	W =180.000 deg,	P =   0.000 deg,	R =    90.000 deg
};
P[5219]{
   GP1:
	UF : 1, UT : 1,		CONFIG : 'N U T, 0, 0, 1',
	X =  91.000  mm,	Y =  97.000  mm,	Z =   0.600 mm,
	W =180.000 deg,	P =   0.000 deg,	R =    90.000 deg
};
P[5220]{
   GP1:
	UF : 1, UT : 1,		CONFIG : 'N U T, 0, 0, 1',
	X =  91.000  mm,	Y =  97.000  mm,	Z =   15.000 mm,
	W =180.000 deg,	P =   0.000 deg,	R =    90.000 deg
};
P[5221]{
   GP1:
	UF : 1, UT : 1,		CONFIG : 'N U T, 0, 0, 1',
	X =  94.000  mm,	Y =  97.000  mm,	Z =   15.000 mm,
	W =180.000 deg,	P =   0.000 deg,	R =    90.000 deg
};
P[5222]{
   GP1:
	UF : 1, UT : 1,		CONFIG : 'N U T, 0, 0, 1',
	X =  94.000  mm,	Y =  97.000  mm,	Z =   0.600 mm,
	W =180.000 deg,	P =   0.000 deg,	R =    90.000 deg
};
P[5223]{
   GP1:
	UF : 1, UT : 1,		CONFIG : 'N U T, 0, 0, 1',
	X =  94.000  mm,	Y =  97.000  mm,	Z =   15.000 mm,
	W =180.000 deg,	P =   0.000 deg,	R =    90.000 deg
};
P[5224]{
   GP1:
	UF : 1, UT : 1,		CONFIG : 'N U T, 0, 0, 1',
	X =  97.000  mm,	Y =  97.000  mm,	Z =   15.000 mm,
	W =180.000 deg,	P =   0.000 deg,	R =    90.000 deg
};
P[5225]{
   GP1:
	UF : 1, UT : 1,		CONFIG : 'N U T, 0, 0, 1',
	X =  97.000  mm,	Y =  97.000  mm,	Z =   0.600 mm,
	W =180.000 deg,	P =   0.000 deg,	R =    90.000 deg
};
P[5226]{
   GP1:
	UF : 1, UT : 1,		CONFIG : 'N U T, 0, 0, 1',
	X =  97.000  mm,	Y =  97.000  mm,	Z =   15.000 mm,
	W =180.000 deg,	P =   0.000 deg,	R =    90.000 deg
};
P[5227]{
   GP1:
	UF : 1, UT : 1,		CONFIG : 'N U T, 0, 0, 1',
	X =  100.000  mm,	Y =  97.000  mm,	Z =   15.000 mm,
	W =180.000 deg,	P =   0.000 deg,	R =    90.000 deg
};
P[5228]{
   GP1:
	UF : 1, UT : 1,		CONFIG : 'N U T, 0, 0, 1',
	X =  100.000  mm,	Y =  97.000  mm,	Z =   0.600 mm,
	W =180.000 deg,	P =   0.000 deg,	R =    90.000 deg
};
P[5229]{
   GP1:
	UF : 1, UT : 1,		CONFIG : 'N U T, 0, 0, 1',
	X =  100.000  mm,	Y =  97.000  mm,	Z =   15.000 mm,
	W =180.000 deg,	P =   0.000 deg,	R =    90.000 deg
};
P[5230]{
   GP1:
	UF : 1, UT : 1,		CONFIG : 'N U T, 0, 0, 1',
	X =  103.000  mm,	Y =  97.000  mm,	Z =   15.000 mm,
	W =180.000 deg,	P =   0.000 deg,	R =    90.000 deg
};
P[5231]{
   GP1:
	UF : 1, UT : 1,		CONFIG : 'N U T, 0, 0, 1',
	X =  103.000  mm,	Y =  97.000  mm,	Z =   0.600 mm,
	W =180.000 deg,	P =   0.000 deg,	R =    90.000 deg
};
P[5232]{
   GP1:
	UF : 1, UT : 1,		CONFIG : 'N U T, 0, 0, 1',
	X =  103.000  mm,	Y =  97.000  mm,	Z =   15.000 mm,
	W =180.000 deg,	P =   0.000 deg,	R =    90.000 deg
};
P[5233]{
   GP1:
	UF : 1, UT : 1,		CONFIG : 'N U T, 0, 0, 1',
	X =  106.000  mm,	Y =  97.000  mm,	Z =   15.000 mm,
	W =180.000 deg,	P =   0.000 deg,	R =    90.000 deg
};
P[5234]{
   GP1:
	UF : 1, UT : 1,		CONFIG : 'N U T, 0, 0, 1',
	X =  106.000  mm,	Y =  97.000  mm,	Z =   0.600 mm,
	W =180.000 deg,	P =   0.000 deg,	R =    90.000 deg
};
P[5235]{
   GP1:
	UF : 1, UT : 1,		CONFIG : 'N U T, 0, 0, 1',
	X =  106.000  mm,	Y =  97.000  mm,	Z =   15.000 mm,
	W =180.000 deg,	P =   0.000 deg,	R =    90.000 deg
};
P[5236]{
   GP1:
	UF : 1, UT : 1,		CONFIG : 'N U T, 0, 0, 1',
	X =  109.000  mm,	Y =  97.000  mm,	Z =   15.000 mm,
	W =180.000 deg,	P =   0.000 deg,	R =    90.000 deg
};
P[5237]{
   GP1:
	UF : 1, UT : 1,		CONFIG : 'N U T, 0, 0, 1',
	X =  109.000  mm,	Y =  97.000  mm,	Z =   0.600 mm,
	W =180.000 deg,	P =   0.000 deg,	R =    90.000 deg
};
P[5238]{
   GP1:
	UF : 1, UT : 1,		CONFIG : 'N U T, 0, 0, 1',
	X =  109.000  mm,	Y =  97.000  mm,	Z =   15.000 mm,
	W =180.000 deg,	P =   0.000 deg,	R =    90.000 deg
};
P[5239]{
   GP1:
	UF : 1, UT : 1,		CONFIG : 'N U T, 0, 0, 1',
	X =  112.000  mm,	Y =  97.000  mm,	Z =   15.000 mm,
	W =180.000 deg,	P =   0.000 deg,	R =    90.000 deg
};
P[5240]{
   GP1:
	UF : 1, UT : 1,		CONFIG : 'N U T, 0, 0, 1',
	X =  112.000  mm,	Y =  97.000  mm,	Z =   0.600 mm,
	W =180.000 deg,	P =   0.000 deg,	R =    90.000 deg
};
P[5241]{
   GP1:
	UF : 1, UT : 1,		CONFIG : 'N U T, 0, 0, 1',
	X =  112.000  mm,	Y =  97.000  mm,	Z =   15.000 mm,
	W =180.000 deg,	P =   0.000 deg,	R =    90.000 deg
};
P[5242]{
   GP1:
	UF : 1, UT : 1,		CONFIG : 'N U T, 0, 0, 1',
	X =  115.000  mm,	Y =  97.000  mm,	Z =   15.000 mm,
	W =180.000 deg,	P =   0.000 deg,	R =    90.000 deg
};
P[5243]{
   GP1:
	UF : 1, UT : 1,		CONFIG : 'N U T, 0, 0, 1',
	X =  115.000  mm,	Y =  97.000  mm,	Z =   0.600 mm,
	W =180.000 deg,	P =   0.000 deg,	R =    90.000 deg
};
P[5244]{
   GP1:
	UF : 1, UT : 1,		CONFIG : 'N U T, 0, 0, 1',
	X =  115.000  mm,	Y =  97.000  mm,	Z =   15.000 mm,
	W =180.000 deg,	P =   0.000 deg,	R =    90.000 deg
};
P[5260]{
   GP1:
	UF : 1, UT : 1,		CONFIG : 'N U T, 0, 0, 1',
	X =  133.000  mm,	Y =  97.000  mm,	Z =   15.000 mm,
	W =180.000 deg,	P =   0.000 deg,	R =    90.000 deg
};
P[5261]{
   GP1:
	UF : 1, UT : 1,		CONFIG : 'N U T, 0, 0, 1',
	X =  133.000  mm,	Y =  97.000  mm,	Z =   0.600 mm,
	W =180.000 deg,	P =   0.000 deg,	R =    90.000 deg
};
P[5262]{
   GP1:
	UF : 1, UT : 1,		CONFIG : 'N U T, 0, 0, 1',
	X =  133.000  mm,	Y =  97.000  mm,	Z =   15.000 mm,
	W =180.000 deg,	P =   0.000 deg,	R =    90.000 deg
};
P[5263]{
   GP1:
	UF : 1, UT : 1,		CONFIG : 'N U T, 0, 0, 1',
	X =  136.000  mm,	Y =  97.000  mm,	Z =   15.000 mm,
	W =180.000 deg,	P =   0.000 deg,	R =    90.000 deg
};
P[5264]{
   GP1:
	UF : 1, UT : 1,		CONFIG : 'N U T, 0, 0, 1',
	X =  136.000  mm,	Y =  97.000  mm,	Z =   0.600 mm,
	W =180.000 deg,	P =   0.000 deg,	R =    90.000 deg
};
P[5265]{
   GP1:
	UF : 1, UT : 1,		CONFIG : 'N U T, 0, 0, 1',
	X =  136.000  mm,	Y =  97.000  mm,	Z =   15.000 mm,
	W =180.000 deg,	P =   0.000 deg,	R =    90.000 deg
};
P[5266]{
   GP1:
	UF : 1, UT : 1,		CONFIG : 'N U T, 0, 0, 1',
	X =  139.000  mm,	Y =  97.000  mm,	Z =   15.000 mm,
	W =180.000 deg,	P =   0.000 deg,	R =    90.000 deg
};
P[5267]{
   GP1:
	UF : 1, UT : 1,		CONFIG : 'N U T, 0, 0, 1',
	X =  139.000  mm,	Y =  97.000  mm,	Z =   0.600 mm,
	W =180.000 deg,	P =   0.000 deg,	R =    90.000 deg
};
P[5268]{
   GP1:
	UF : 1, UT : 1,		CONFIG : 'N U T, 0, 0, 1',
	X =  139.000  mm,	Y =  97.000  mm,	Z =   15.000 mm,
	W =180.000 deg,	P =   0.000 deg,	R =    90.000 deg
};
P[5278]{
   GP1:
	UF : 1, UT : 1,		CONFIG : 'N U T, 0, 0, 1',
	X =  163.000  mm,	Y =  97.000  mm,	Z =   15.000 mm,
	W =180.000 deg,	P =   0.000 deg,	R =    90.000 deg
};
P[5279]{
   GP1:
	UF : 1, UT : 1,		CONFIG : 'N U T, 0, 0, 1',
	X =  163.000  mm,	Y =  97.000  mm,	Z =   0.600 mm,
	W =180.000 deg,	P =   0.000 deg,	R =    90.000 deg
};
P[5280]{
   GP1:
	UF : 1, UT : 1,		CONFIG : 'N U T, 0, 0, 1',
	X =  163.000  mm,	Y =  97.000  mm,	Z =   15.000 mm,
	W =180.000 deg,	P =   0.000 deg,	R =    90.000 deg
};
P[5281]{
   GP1:
	UF : 1, UT : 1,		CONFIG : 'N U T, 0, 0, 1',
	X =  166.000  mm,	Y =  97.000  mm,	Z =   15.000 mm,
	W =180.000 deg,	P =   0.000 deg,	R =    90.000 deg
};
P[5282]{
   GP1:
	UF : 1, UT : 1,		CONFIG : 'N U T, 0, 0, 1',
	X =  166.000  mm,	Y =  97.000  mm,	Z =   0.600 mm,
	W =180.000 deg,	P =   0.000 deg,	R =    90.000 deg
};
P[5283]{
   GP1:
	UF : 1, UT : 1,		CONFIG : 'N U T, 0, 0, 1',
	X =  166.000  mm,	Y =  97.000  mm,	Z =   15.000 mm,
	W =180.000 deg,	P =   0.000 deg,	R =    90.000 deg
};
P[5284]{
   GP1:
	UF : 1, UT : 1,		CONFIG : 'N U T, 0, 0, 1',
	X =  169.000  mm,	Y =  97.000  mm,	Z =   15.000 mm,
	W =180.000 deg,	P =   0.000 deg,	R =    90.000 deg
};
P[5285]{
   GP1:
	UF : 1, UT : 1,		CONFIG : 'N U T, 0, 0, 1',
	X =  169.000  mm,	Y =  97.000  mm,	Z =   0.600 mm,
	W =180.000 deg,	P =   0.000 deg,	R =    90.000 deg
};
P[5286]{
   GP1:
	UF : 1, UT : 1,		CONFIG : 'N U T, 0, 0, 1',
	X =  169.000  mm,	Y =  97.000  mm,	Z =   15.000 mm,
	W =180.000 deg,	P =   0.000 deg,	R =    90.000 deg
};
P[5287]{
   GP1:
	UF : 1, UT : 1,		CONFIG : 'N U T, 0, 0, 1',
	X =  172.000  mm,	Y =  97.000  mm,	Z =   15.000 mm,
	W =180.000 deg,	P =   0.000 deg,	R =    90.000 deg
};
P[5288]{
   GP1:
	UF : 1, UT : 1,		CONFIG : 'N U T, 0, 0, 1',
	X =  172.000  mm,	Y =  97.000  mm,	Z =   0.600 mm,
	W =180.000 deg,	P =   0.000 deg,	R =    90.000 deg
};
P[5289]{
   GP1:
	UF : 1, UT : 1,		CONFIG : 'N U T, 0, 0, 1',
	X =  172.000  mm,	Y =  97.000  mm,	Z =   15.000 mm,
	W =180.000 deg,	P =   0.000 deg,	R =    90.000 deg
};
P[5290]{
   GP1:
	UF : 1, UT : 1,		CONFIG : 'N U T, 0, 0, 1',
	X =  175.000  mm,	Y =  97.000  mm,	Z =   15.000 mm,
	W =180.000 deg,	P =   0.000 deg,	R =    90.000 deg
};
P[5291]{
   GP1:
	UF : 1, UT : 1,		CONFIG : 'N U T, 0, 0, 1',
	X =  175.000  mm,	Y =  97.000  mm,	Z =   0.600 mm,
	W =180.000 deg,	P =   0.000 deg,	R =    90.000 deg
};
P[5292]{
   GP1:
	UF : 1, UT : 1,		CONFIG : 'N U T, 0, 0, 1',
	X =  175.000  mm,	Y =  97.000  mm,	Z =   15.000 mm,
	W =180.000 deg,	P =   0.000 deg,	R =    90.000 deg
};
P[5293]{
   GP1:
	UF : 1, UT : 1,		CONFIG : 'N U T, 0, 0, 1',
	X =  178.000  mm,	Y =  97.000  mm,	Z =   15.000 mm,
	W =180.000 deg,	P =   0.000 deg,	R =    90.000 deg
};
P[5294]{
   GP1:
	UF : 1, UT : 1,		CONFIG : 'N U T, 0, 0, 1',
	X =  178.000  mm,	Y =  97.000  mm,	Z =   0.600 mm,
	W =180.000 deg,	P =   0.000 deg,	R =    90.000 deg
};
P[5295]{
   GP1:
	UF : 1, UT : 1,		CONFIG : 'N U T, 0, 0, 1',
	X =  178.000  mm,	Y =  97.000  mm,	Z =   15.000 mm,
	W =180.000 deg,	P =   0.000 deg,	R =    90.000 deg
};
P[5299]{
   GP1:
	UF : 1, UT : 1,		CONFIG : 'N U T, 0, 0, 1',
	X =  4.000  mm,	Y =  100.000  mm,	Z =   15.000 mm,
	W =180.000 deg,	P =   0.000 deg,	R =    90.000 deg
};
P[5300]{
   GP1:
	UF : 1, UT : 1,		CONFIG : 'N U T, 0, 0, 1',
	X =  4.000  mm,	Y =  100.000  mm,	Z =   0.600 mm,
	W =180.000 deg,	P =   0.000 deg,	R =    90.000 deg
};
P[5301]{
   GP1:
	UF : 1, UT : 1,		CONFIG : 'N U T, 0, 0, 1',
	X =  4.000  mm,	Y =  100.000  mm,	Z =   15.000 mm,
	W =180.000 deg,	P =   0.000 deg,	R =    90.000 deg
};
P[5305]{
   GP1:
	UF : 1, UT : 1,		CONFIG : 'N U T, 0, 0, 1',
	X =  10.000  mm,	Y =  100.000  mm,	Z =   15.000 mm,
	W =180.000 deg,	P =   0.000 deg,	R =    90.000 deg
};
P[5306]{
   GP1:
	UF : 1, UT : 1,		CONFIG : 'N U T, 0, 0, 1',
	X =  10.000  mm,	Y =  100.000  mm,	Z =   0.600 mm,
	W =180.000 deg,	P =   0.000 deg,	R =    90.000 deg
};
P[5307]{
   GP1:
	UF : 1, UT : 1,		CONFIG : 'N U T, 0, 0, 1',
	X =  10.000  mm,	Y =  100.000  mm,	Z =   15.000 mm,
	W =180.000 deg,	P =   0.000 deg,	R =    90.000 deg
};
P[5308]{
   GP1:
	UF : 1, UT : 1,		CONFIG : 'N U T, 0, 0, 1',
	X =  13.000  mm,	Y =  100.000  mm,	Z =   15.000 mm,
	W =180.000 deg,	P =   0.000 deg,	R =    90.000 deg
};
P[5309]{
   GP1:
	UF : 1, UT : 1,		CONFIG : 'N U T, 0, 0, 1',
	X =  13.000  mm,	Y =  100.000  mm,	Z =   0.600 mm,
	W =180.000 deg,	P =   0.000 deg,	R =    90.000 deg
};
P[5310]{
   GP1:
	UF : 1, UT : 1,		CONFIG : 'N U T, 0, 0, 1',
	X =  13.000  mm,	Y =  100.000  mm,	Z =   15.000 mm,
	W =180.000 deg,	P =   0.000 deg,	R =    90.000 deg
};
P[5320]{
   GP1:
	UF : 1, UT : 1,		CONFIG : 'N U T, 0, 0, 1',
	X =  25.000  mm,	Y =  100.000  mm,	Z =   15.000 mm,
	W =180.000 deg,	P =   0.000 deg,	R =    90.000 deg
};
P[5321]{
   GP1:
	UF : 1, UT : 1,		CONFIG : 'N U T, 0, 0, 1',
	X =  25.000  mm,	Y =  100.000  mm,	Z =   0.600 mm,
	W =180.000 deg,	P =   0.000 deg,	R =    90.000 deg
};
P[5322]{
   GP1:
	UF : 1, UT : 1,		CONFIG : 'N U T, 0, 0, 1',
	X =  25.000  mm,	Y =  100.000  mm,	Z =   15.000 mm,
	W =180.000 deg,	P =   0.000 deg,	R =    90.000 deg
};
P[5323]{
   GP1:
	UF : 1, UT : 1,		CONFIG : 'N U T, 0, 0, 1',
	X =  28.000  mm,	Y =  100.000  mm,	Z =   15.000 mm,
	W =180.000 deg,	P =   0.000 deg,	R =    90.000 deg
};
P[5324]{
   GP1:
	UF : 1, UT : 1,		CONFIG : 'N U T, 0, 0, 1',
	X =  28.000  mm,	Y =  100.000  mm,	Z =   0.600 mm,
	W =180.000 deg,	P =   0.000 deg,	R =    90.000 deg
};
P[5325]{
   GP1:
	UF : 1, UT : 1,		CONFIG : 'N U T, 0, 0, 1',
	X =  28.000  mm,	Y =  100.000  mm,	Z =   15.000 mm,
	W =180.000 deg,	P =   0.000 deg,	R =    90.000 deg
};
P[5335]{
   GP1:
	UF : 1, UT : 1,		CONFIG : 'N U T, 0, 0, 1',
	X =  40.000  mm,	Y =  100.000  mm,	Z =   15.000 mm,
	W =180.000 deg,	P =   0.000 deg,	R =    90.000 deg
};
P[5336]{
   GP1:
	UF : 1, UT : 1,		CONFIG : 'N U T, 0, 0, 1',
	X =  40.000  mm,	Y =  100.000  mm,	Z =   0.600 mm,
	W =180.000 deg,	P =   0.000 deg,	R =    90.000 deg
};
P[5337]{
   GP1:
	UF : 1, UT : 1,		CONFIG : 'N U T, 0, 0, 1',
	X =  40.000  mm,	Y =  100.000  mm,	Z =   15.000 mm,
	W =180.000 deg,	P =   0.000 deg,	R =    90.000 deg
};
P[5338]{
   GP1:
	UF : 1, UT : 1,		CONFIG : 'N U T, 0, 0, 1',
	X =  43.000  mm,	Y =  100.000  mm,	Z =   15.000 mm,
	W =180.000 deg,	P =   0.000 deg,	R =    90.000 deg
};
P[5339]{
   GP1:
	UF : 1, UT : 1,		CONFIG : 'N U T, 0, 0, 1',
	X =  43.000  mm,	Y =  100.000  mm,	Z =   0.600 mm,
	W =180.000 deg,	P =   0.000 deg,	R =    90.000 deg
};
P[5340]{
   GP1:
	UF : 1, UT : 1,		CONFIG : 'N U T, 0, 0, 1',
	X =  43.000  mm,	Y =  100.000  mm,	Z =   15.000 mm,
	W =180.000 deg,	P =   0.000 deg,	R =    90.000 deg
};
P[5341]{
   GP1:
	UF : 1, UT : 1,		CONFIG : 'N U T, 0, 0, 1',
	X =  46.000  mm,	Y =  100.000  mm,	Z =   15.000 mm,
	W =180.000 deg,	P =   0.000 deg,	R =    90.000 deg
};
P[5342]{
   GP1:
	UF : 1, UT : 1,		CONFIG : 'N U T, 0, 0, 1',
	X =  46.000  mm,	Y =  100.000  mm,	Z =   0.600 mm,
	W =180.000 deg,	P =   0.000 deg,	R =    90.000 deg
};
P[5343]{
   GP1:
	UF : 1, UT : 1,		CONFIG : 'N U T, 0, 0, 1',
	X =  46.000  mm,	Y =  100.000  mm,	Z =   15.000 mm,
	W =180.000 deg,	P =   0.000 deg,	R =    90.000 deg
};
P[5344]{
   GP1:
	UF : 1, UT : 1,		CONFIG : 'N U T, 0, 0, 1',
	X =  49.000  mm,	Y =  100.000  mm,	Z =   15.000 mm,
	W =180.000 deg,	P =   0.000 deg,	R =    90.000 deg
};
P[5345]{
   GP1:
	UF : 1, UT : 1,		CONFIG : 'N U T, 0, 0, 1',
	X =  49.000  mm,	Y =  100.000  mm,	Z =   0.600 mm,
	W =180.000 deg,	P =   0.000 deg,	R =    90.000 deg
};
P[5346]{
   GP1:
	UF : 1, UT : 1,		CONFIG : 'N U T, 0, 0, 1',
	X =  49.000  mm,	Y =  100.000  mm,	Z =   15.000 mm,
	W =180.000 deg,	P =   0.000 deg,	R =    90.000 deg
};
P[5347]{
   GP1:
	UF : 1, UT : 1,		CONFIG : 'N U T, 0, 0, 1',
	X =  52.000  mm,	Y =  100.000  mm,	Z =   15.000 mm,
	W =180.000 deg,	P =   0.000 deg,	R =    90.000 deg
};
P[5348]{
   GP1:
	UF : 1, UT : 1,		CONFIG : 'N U T, 0, 0, 1',
	X =  52.000  mm,	Y =  100.000  mm,	Z =   0.600 mm,
	W =180.000 deg,	P =   0.000 deg,	R =    90.000 deg
};
P[5349]{
   GP1:
	UF : 1, UT : 1,		CONFIG : 'N U T, 0, 0, 1',
	X =  52.000  mm,	Y =  100.000  mm,	Z =   15.000 mm,
	W =180.000 deg,	P =   0.000 deg,	R =    90.000 deg
};
P[5350]{
   GP1:
	UF : 1, UT : 1,		CONFIG : 'N U T, 0, 0, 1',
	X =  55.000  mm,	Y =  100.000  mm,	Z =   15.000 mm,
	W =180.000 deg,	P =   0.000 deg,	R =    90.000 deg
};
P[5351]{
   GP1:
	UF : 1, UT : 1,		CONFIG : 'N U T, 0, 0, 1',
	X =  55.000  mm,	Y =  100.000  mm,	Z =   0.600 mm,
	W =180.000 deg,	P =   0.000 deg,	R =    90.000 deg
};
P[5352]{
   GP1:
	UF : 1, UT : 1,		CONFIG : 'N U T, 0, 0, 1',
	X =  55.000  mm,	Y =  100.000  mm,	Z =   15.000 mm,
	W =180.000 deg,	P =   0.000 deg,	R =    90.000 deg
};
P[5356]{
   GP1:
	UF : 1, UT : 1,		CONFIG : 'N U T, 0, 0, 1',
	X =  61.000  mm,	Y =  100.000  mm,	Z =   15.000 mm,
	W =180.000 deg,	P =   0.000 deg,	R =    90.000 deg
};
P[5357]{
   GP1:
	UF : 1, UT : 1,		CONFIG : 'N U T, 0, 0, 1',
	X =  61.000  mm,	Y =  100.000  mm,	Z =   0.600 mm,
	W =180.000 deg,	P =   0.000 deg,	R =    90.000 deg
};
P[5358]{
   GP1:
	UF : 1, UT : 1,		CONFIG : 'N U T, 0, 0, 1',
	X =  61.000  mm,	Y =  100.000  mm,	Z =   15.000 mm,
	W =180.000 deg,	P =   0.000 deg,	R =    90.000 deg
};
P[5386]{
   GP1:
	UF : 1, UT : 1,		CONFIG : 'N U T, 0, 0, 1',
	X =  91.000  mm,	Y =  100.000  mm,	Z =   15.000 mm,
	W =180.000 deg,	P =   0.000 deg,	R =    90.000 deg
};
P[5387]{
   GP1:
	UF : 1, UT : 1,		CONFIG : 'N U T, 0, 0, 1',
	X =  91.000  mm,	Y =  100.000  mm,	Z =   0.600 mm,
	W =180.000 deg,	P =   0.000 deg,	R =    90.000 deg
};
P[5388]{
   GP1:
	UF : 1, UT : 1,		CONFIG : 'N U T, 0, 0, 1',
	X =  91.000  mm,	Y =  100.000  mm,	Z =   15.000 mm,
	W =180.000 deg,	P =   0.000 deg,	R =    90.000 deg
};
P[5389]{
   GP1:
	UF : 1, UT : 1,		CONFIG : 'N U T, 0, 0, 1',
	X =  94.000  mm,	Y =  100.000  mm,	Z =   15.000 mm,
	W =180.000 deg,	P =   0.000 deg,	R =    90.000 deg
};
P[5390]{
   GP1:
	UF : 1, UT : 1,		CONFIG : 'N U T, 0, 0, 1',
	X =  94.000  mm,	Y =  100.000  mm,	Z =   0.600 mm,
	W =180.000 deg,	P =   0.000 deg,	R =    90.000 deg
};
P[5391]{
   GP1:
	UF : 1, UT : 1,		CONFIG : 'N U T, 0, 0, 1',
	X =  94.000  mm,	Y =  100.000  mm,	Z =   15.000 mm,
	W =180.000 deg,	P =   0.000 deg,	R =    90.000 deg
};
P[5392]{
   GP1:
	UF : 1, UT : 1,		CONFIG : 'N U T, 0, 0, 1',
	X =  97.000  mm,	Y =  100.000  mm,	Z =   15.000 mm,
	W =180.000 deg,	P =   0.000 deg,	R =    90.000 deg
};
P[5393]{
   GP1:
	UF : 1, UT : 1,		CONFIG : 'N U T, 0, 0, 1',
	X =  97.000  mm,	Y =  100.000  mm,	Z =   0.600 mm,
	W =180.000 deg,	P =   0.000 deg,	R =    90.000 deg
};
P[5394]{
   GP1:
	UF : 1, UT : 1,		CONFIG : 'N U T, 0, 0, 1',
	X =  97.000  mm,	Y =  100.000  mm,	Z =   15.000 mm,
	W =180.000 deg,	P =   0.000 deg,	R =    90.000 deg
};
P[5395]{
   GP1:
	UF : 1, UT : 1,		CONFIG : 'N U T, 0, 0, 1',
	X =  100.000  mm,	Y =  100.000  mm,	Z =   15.000 mm,
	W =180.000 deg,	P =   0.000 deg,	R =    90.000 deg
};
P[5396]{
   GP1:
	UF : 1, UT : 1,		CONFIG : 'N U T, 0, 0, 1',
	X =  100.000  mm,	Y =  100.000  mm,	Z =   0.600 mm,
	W =180.000 deg,	P =   0.000 deg,	R =    90.000 deg
};
P[5397]{
   GP1:
	UF : 1, UT : 1,		CONFIG : 'N U T, 0, 0, 1',
	X =  100.000  mm,	Y =  100.000  mm,	Z =   15.000 mm,
	W =180.000 deg,	P =   0.000 deg,	R =    90.000 deg
};
P[5398]{
   GP1:
	UF : 1, UT : 1,		CONFIG : 'N U T, 0, 0, 1',
	X =  103.000  mm,	Y =  100.000  mm,	Z =   15.000 mm,
	W =180.000 deg,	P =   0.000 deg,	R =    90.000 deg
};
P[5399]{
   GP1:
	UF : 1, UT : 1,		CONFIG : 'N U T, 0, 0, 1',
	X =  103.000  mm,	Y =  100.000  mm,	Z =   0.600 mm,
	W =180.000 deg,	P =   0.000 deg,	R =    90.000 deg
};
P[5400]{
   GP1:
	UF : 1, UT : 1,		CONFIG : 'N U T, 0, 0, 1',
	X =  103.000  mm,	Y =  100.000  mm,	Z =   15.000 mm,
	W =180.000 deg,	P =   0.000 deg,	R =    90.000 deg
};
P[5401]{
   GP1:
	UF : 1, UT : 1,		CONFIG : 'N U T, 0, 0, 1',
	X =  106.000  mm,	Y =  100.000  mm,	Z =   15.000 mm,
	W =180.000 deg,	P =   0.000 deg,	R =    90.000 deg
};
P[5402]{
   GP1:
	UF : 1, UT : 1,		CONFIG : 'N U T, 0, 0, 1',
	X =  106.000  mm,	Y =  100.000  mm,	Z =   0.600 mm,
	W =180.000 deg,	P =   0.000 deg,	R =    90.000 deg
};
P[5403]{
   GP1:
	UF : 1, UT : 1,		CONFIG : 'N U T, 0, 0, 1',
	X =  106.000  mm,	Y =  100.000  mm,	Z =   15.000 mm,
	W =180.000 deg,	P =   0.000 deg,	R =    90.000 deg
};
P[5404]{
   GP1:
	UF : 1, UT : 1,		CONFIG : 'N U T, 0, 0, 1',
	X =  109.000  mm,	Y =  100.000  mm,	Z =   15.000 mm,
	W =180.000 deg,	P =   0.000 deg,	R =    90.000 deg
};
P[5405]{
   GP1:
	UF : 1, UT : 1,		CONFIG : 'N U T, 0, 0, 1',
	X =  109.000  mm,	Y =  100.000  mm,	Z =   0.600 mm,
	W =180.000 deg,	P =   0.000 deg,	R =    90.000 deg
};
P[5406]{
   GP1:
	UF : 1, UT : 1,		CONFIG : 'N U T, 0, 0, 1',
	X =  109.000  mm,	Y =  100.000  mm,	Z =   15.000 mm,
	W =180.000 deg,	P =   0.000 deg,	R =    90.000 deg
};
P[5407]{
   GP1:
	UF : 1, UT : 1,		CONFIG : 'N U T, 0, 0, 1',
	X =  112.000  mm,	Y =  100.000  mm,	Z =   15.000 mm,
	W =180.000 deg,	P =   0.000 deg,	R =    90.000 deg
};
P[5408]{
   GP1:
	UF : 1, UT : 1,		CONFIG : 'N U T, 0, 0, 1',
	X =  112.000  mm,	Y =  100.000  mm,	Z =   0.600 mm,
	W =180.000 deg,	P =   0.000 deg,	R =    90.000 deg
};
P[5409]{
   GP1:
	UF : 1, UT : 1,		CONFIG : 'N U T, 0, 0, 1',
	X =  112.000  mm,	Y =  100.000  mm,	Z =   15.000 mm,
	W =180.000 deg,	P =   0.000 deg,	R =    90.000 deg
};
P[5410]{
   GP1:
	UF : 1, UT : 1,		CONFIG : 'N U T, 0, 0, 1',
	X =  115.000  mm,	Y =  100.000  mm,	Z =   15.000 mm,
	W =180.000 deg,	P =   0.000 deg,	R =    90.000 deg
};
P[5411]{
   GP1:
	UF : 1, UT : 1,		CONFIG : 'N U T, 0, 0, 1',
	X =  115.000  mm,	Y =  100.000  mm,	Z =   0.600 mm,
	W =180.000 deg,	P =   0.000 deg,	R =    90.000 deg
};
P[5412]{
   GP1:
	UF : 1, UT : 1,		CONFIG : 'N U T, 0, 0, 1',
	X =  115.000  mm,	Y =  100.000  mm,	Z =   15.000 mm,
	W =180.000 deg,	P =   0.000 deg,	R =    90.000 deg
};
P[5413]{
   GP1:
	UF : 1, UT : 1,		CONFIG : 'N U T, 0, 0, 1',
	X =  118.000  mm,	Y =  100.000  mm,	Z =   15.000 mm,
	W =180.000 deg,	P =   0.000 deg,	R =    90.000 deg
};
P[5414]{
   GP1:
	UF : 1, UT : 1,		CONFIG : 'N U T, 0, 0, 1',
	X =  118.000  mm,	Y =  100.000  mm,	Z =   0.600 mm,
	W =180.000 deg,	P =   0.000 deg,	R =    90.000 deg
};
P[5415]{
   GP1:
	UF : 1, UT : 1,		CONFIG : 'N U T, 0, 0, 1',
	X =  118.000  mm,	Y =  100.000  mm,	Z =   15.000 mm,
	W =180.000 deg,	P =   0.000 deg,	R =    90.000 deg
};
P[5428]{
   GP1:
	UF : 1, UT : 1,		CONFIG : 'N U T, 0, 0, 1',
	X =  133.000  mm,	Y =  100.000  mm,	Z =   15.000 mm,
	W =180.000 deg,	P =   0.000 deg,	R =    90.000 deg
};
P[5429]{
   GP1:
	UF : 1, UT : 1,		CONFIG : 'N U T, 0, 0, 1',
	X =  133.000  mm,	Y =  100.000  mm,	Z =   0.600 mm,
	W =180.000 deg,	P =   0.000 deg,	R =    90.000 deg
};
P[5430]{
   GP1:
	UF : 1, UT : 1,		CONFIG : 'N U T, 0, 0, 1',
	X =  133.000  mm,	Y =  100.000  mm,	Z =   15.000 mm,
	W =180.000 deg,	P =   0.000 deg,	R =    90.000 deg
};
P[5431]{
   GP1:
	UF : 1, UT : 1,		CONFIG : 'N U T, 0, 0, 1',
	X =  136.000  mm,	Y =  100.000  mm,	Z =   15.000 mm,
	W =180.000 deg,	P =   0.000 deg,	R =    90.000 deg
};
P[5432]{
   GP1:
	UF : 1, UT : 1,		CONFIG : 'N U T, 0, 0, 1',
	X =  136.000  mm,	Y =  100.000  mm,	Z =   0.600 mm,
	W =180.000 deg,	P =   0.000 deg,	R =    90.000 deg
};
P[5433]{
   GP1:
	UF : 1, UT : 1,		CONFIG : 'N U T, 0, 0, 1',
	X =  136.000  mm,	Y =  100.000  mm,	Z =   15.000 mm,
	W =180.000 deg,	P =   0.000 deg,	R =    90.000 deg
};
P[5434]{
   GP1:
	UF : 1, UT : 1,		CONFIG : 'N U T, 0, 0, 1',
	X =  139.000  mm,	Y =  100.000  mm,	Z =   15.000 mm,
	W =180.000 deg,	P =   0.000 deg,	R =    90.000 deg
};
P[5435]{
   GP1:
	UF : 1, UT : 1,		CONFIG : 'N U T, 0, 0, 1',
	X =  139.000  mm,	Y =  100.000  mm,	Z =   0.600 mm,
	W =180.000 deg,	P =   0.000 deg,	R =    90.000 deg
};
P[5436]{
   GP1:
	UF : 1, UT : 1,		CONFIG : 'N U T, 0, 0, 1',
	X =  139.000  mm,	Y =  100.000  mm,	Z =   15.000 mm,
	W =180.000 deg,	P =   0.000 deg,	R =    90.000 deg
};
P[5437]{
   GP1:
	UF : 1, UT : 1,		CONFIG : 'N U T, 0, 0, 1',
	X =  142.000  mm,	Y =  100.000  mm,	Z =   15.000 mm,
	W =180.000 deg,	P =   0.000 deg,	R =    90.000 deg
};
P[5438]{
   GP1:
	UF : 1, UT : 1,		CONFIG : 'N U T, 0, 0, 1',
	X =  142.000  mm,	Y =  100.000  mm,	Z =   0.600 mm,
	W =180.000 deg,	P =   0.000 deg,	R =    90.000 deg
};
P[5439]{
   GP1:
	UF : 1, UT : 1,		CONFIG : 'N U T, 0, 0, 1',
	X =  142.000  mm,	Y =  100.000  mm,	Z =   15.000 mm,
	W =180.000 deg,	P =   0.000 deg,	R =    90.000 deg
};
P[5446]{
   GP1:
	UF : 1, UT : 1,		CONFIG : 'N U T, 0, 0, 1',
	X =  163.000  mm,	Y =  100.000  mm,	Z =   15.000 mm,
	W =180.000 deg,	P =   0.000 deg,	R =    90.000 deg
};
P[5447]{
   GP1:
	UF : 1, UT : 1,		CONFIG : 'N U T, 0, 0, 1',
	X =  163.000  mm,	Y =  100.000  mm,	Z =   0.600 mm,
	W =180.000 deg,	P =   0.000 deg,	R =    90.000 deg
};
P[5448]{
   GP1:
	UF : 1, UT : 1,		CONFIG : 'N U T, 0, 0, 1',
	X =  163.000  mm,	Y =  100.000  mm,	Z =   15.000 mm,
	W =180.000 deg,	P =   0.000 deg,	R =    90.000 deg
};
P[5449]{
   GP1:
	UF : 1, UT : 1,		CONFIG : 'N U T, 0, 0, 1',
	X =  166.000  mm,	Y =  100.000  mm,	Z =   15.000 mm,
	W =180.000 deg,	P =   0.000 deg,	R =    90.000 deg
};
P[5450]{
   GP1:
	UF : 1, UT : 1,		CONFIG : 'N U T, 0, 0, 1',
	X =  166.000  mm,	Y =  100.000  mm,	Z =   0.600 mm,
	W =180.000 deg,	P =   0.000 deg,	R =    90.000 deg
};
P[5451]{
   GP1:
	UF : 1, UT : 1,		CONFIG : 'N U T, 0, 0, 1',
	X =  166.000  mm,	Y =  100.000  mm,	Z =   15.000 mm,
	W =180.000 deg,	P =   0.000 deg,	R =    90.000 deg
};
P[5452]{
   GP1:
	UF : 1, UT : 1,		CONFIG : 'N U T, 0, 0, 1',
	X =  169.000  mm,	Y =  100.000  mm,	Z =   15.000 mm,
	W =180.000 deg,	P =   0.000 deg,	R =    90.000 deg
};
P[5453]{
   GP1:
	UF : 1, UT : 1,		CONFIG : 'N U T, 0, 0, 1',
	X =  169.000  mm,	Y =  100.000  mm,	Z =   0.600 mm,
	W =180.000 deg,	P =   0.000 deg,	R =    90.000 deg
};
P[5454]{
   GP1:
	UF : 1, UT : 1,		CONFIG : 'N U T, 0, 0, 1',
	X =  169.000  mm,	Y =  100.000  mm,	Z =   15.000 mm,
	W =180.000 deg,	P =   0.000 deg,	R =    90.000 deg
};
P[5455]{
   GP1:
	UF : 1, UT : 1,		CONFIG : 'N U T, 0, 0, 1',
	X =  172.000  mm,	Y =  100.000  mm,	Z =   15.000 mm,
	W =180.000 deg,	P =   0.000 deg,	R =    90.000 deg
};
P[5456]{
   GP1:
	UF : 1, UT : 1,		CONFIG : 'N U T, 0, 0, 1',
	X =  172.000  mm,	Y =  100.000  mm,	Z =   0.600 mm,
	W =180.000 deg,	P =   0.000 deg,	R =    90.000 deg
};
P[5457]{
   GP1:
	UF : 1, UT : 1,		CONFIG : 'N U T, 0, 0, 1',
	X =  172.000  mm,	Y =  100.000  mm,	Z =   15.000 mm,
	W =180.000 deg,	P =   0.000 deg,	R =    90.000 deg
};
P[5458]{
   GP1:
	UF : 1, UT : 1,		CONFIG : 'N U T, 0, 0, 1',
	X =  175.000  mm,	Y =  100.000  mm,	Z =   15.000 mm,
	W =180.000 deg,	P =   0.000 deg,	R =    90.000 deg
};
P[5459]{
   GP1:
	UF : 1, UT : 1,		CONFIG : 'N U T, 0, 0, 1',
	X =  175.000  mm,	Y =  100.000  mm,	Z =   0.600 mm,
	W =180.000 deg,	P =   0.000 deg,	R =    90.000 deg
};
P[5460]{
   GP1:
	UF : 1, UT : 1,		CONFIG : 'N U T, 0, 0, 1',
	X =  175.000  mm,	Y =  100.000  mm,	Z =   15.000 mm,
	W =180.000 deg,	P =   0.000 deg,	R =    90.000 deg
};
P[5461]{
   GP1:
	UF : 1, UT : 1,		CONFIG : 'N U T, 0, 0, 1',
	X =  178.000  mm,	Y =  100.000  mm,	Z =   15.000 mm,
	W =180.000 deg,	P =   0.000 deg,	R =    90.000 deg
};
P[5462]{
   GP1:
	UF : 1, UT : 1,		CONFIG : 'N U T, 0, 0, 1',
	X =  178.000  mm,	Y =  100.000  mm,	Z =   0.600 mm,
	W =180.000 deg,	P =   0.000 deg,	R =    90.000 deg
};
P[5463]{
   GP1:
	UF : 1, UT : 1,		CONFIG : 'N U T, 0, 0, 1',
	X =  178.000  mm,	Y =  100.000  mm,	Z =   15.000 mm,
	W =180.000 deg,	P =   0.000 deg,	R =    90.000 deg
};
P[5467]{
   GP1:
	UF : 1, UT : 1,		CONFIG : 'N U T, 0, 0, 1',
	X =  4.000  mm,	Y =  103.000  mm,	Z =   15.000 mm,
	W =180.000 deg,	P =   0.000 deg,	R =    90.000 deg
};
P[5468]{
   GP1:
	UF : 1, UT : 1,		CONFIG : 'N U T, 0, 0, 1',
	X =  4.000  mm,	Y =  103.000  mm,	Z =   0.600 mm,
	W =180.000 deg,	P =   0.000 deg,	R =    90.000 deg
};
P[5469]{
   GP1:
	UF : 1, UT : 1,		CONFIG : 'N U T, 0, 0, 1',
	X =  4.000  mm,	Y =  103.000  mm,	Z =   15.000 mm,
	W =180.000 deg,	P =   0.000 deg,	R =    90.000 deg
};
P[5470]{
   GP1:
	UF : 1, UT : 1,		CONFIG : 'N U T, 0, 0, 1',
	X =  7.000  mm,	Y =  103.000  mm,	Z =   15.000 mm,
	W =180.000 deg,	P =   0.000 deg,	R =    90.000 deg
};
P[5471]{
   GP1:
	UF : 1, UT : 1,		CONFIG : 'N U T, 0, 0, 1',
	X =  7.000  mm,	Y =  103.000  mm,	Z =   0.600 mm,
	W =180.000 deg,	P =   0.000 deg,	R =    90.000 deg
};
P[5472]{
   GP1:
	UF : 1, UT : 1,		CONFIG : 'N U T, 0, 0, 1',
	X =  7.000  mm,	Y =  103.000  mm,	Z =   15.000 mm,
	W =180.000 deg,	P =   0.000 deg,	R =    90.000 deg
};
P[5476]{
   GP1:
	UF : 1, UT : 1,		CONFIG : 'N U T, 0, 0, 1',
	X =  13.000  mm,	Y =  103.000  mm,	Z =   15.000 mm,
	W =180.000 deg,	P =   0.000 deg,	R =    90.000 deg
};
P[5477]{
   GP1:
	UF : 1, UT : 1,		CONFIG : 'N U T, 0, 0, 1',
	X =  13.000  mm,	Y =  103.000  mm,	Z =   0.600 mm,
	W =180.000 deg,	P =   0.000 deg,	R =    90.000 deg
};
P[5478]{
   GP1:
	UF : 1, UT : 1,		CONFIG : 'N U T, 0, 0, 1',
	X =  13.000  mm,	Y =  103.000  mm,	Z =   15.000 mm,
	W =180.000 deg,	P =   0.000 deg,	R =    90.000 deg
};
P[5509]{
   GP1:
	UF : 1, UT : 1,		CONFIG : 'N U T, 0, 0, 1',
	X =  46.000  mm,	Y =  103.000  mm,	Z =   15.000 mm,
	W =180.000 deg,	P =   0.000 deg,	R =    90.000 deg
};
P[5510]{
   GP1:
	UF : 1, UT : 1,		CONFIG : 'N U T, 0, 0, 1',
	X =  46.000  mm,	Y =  103.000  mm,	Z =   0.600 mm,
	W =180.000 deg,	P =   0.000 deg,	R =    90.000 deg
};
P[5511]{
   GP1:
	UF : 1, UT : 1,		CONFIG : 'N U T, 0, 0, 1',
	X =  46.000  mm,	Y =  103.000  mm,	Z =   15.000 mm,
	W =180.000 deg,	P =   0.000 deg,	R =    90.000 deg
};
P[5512]{
   GP1:
	UF : 1, UT : 1,		CONFIG : 'N U T, 0, 0, 1',
	X =  49.000  mm,	Y =  103.000  mm,	Z =   15.000 mm,
	W =180.000 deg,	P =   0.000 deg,	R =    90.000 deg
};
P[5513]{
   GP1:
	UF : 1, UT : 1,		CONFIG : 'N U T, 0, 0, 1',
	X =  49.000  mm,	Y =  103.000  mm,	Z =   0.600 mm,
	W =180.000 deg,	P =   0.000 deg,	R =    90.000 deg
};
P[5514]{
   GP1:
	UF : 1, UT : 1,		CONFIG : 'N U T, 0, 0, 1',
	X =  49.000  mm,	Y =  103.000  mm,	Z =   15.000 mm,
	W =180.000 deg,	P =   0.000 deg,	R =    90.000 deg
};
P[5515]{
   GP1:
	UF : 1, UT : 1,		CONFIG : 'N U T, 0, 0, 1',
	X =  52.000  mm,	Y =  103.000  mm,	Z =   15.000 mm,
	W =180.000 deg,	P =   0.000 deg,	R =    90.000 deg
};
P[5516]{
   GP1:
	UF : 1, UT : 1,		CONFIG : 'N U T, 0, 0, 1',
	X =  52.000  mm,	Y =  103.000  mm,	Z =   0.600 mm,
	W =180.000 deg,	P =   0.000 deg,	R =    90.000 deg
};
P[5517]{
   GP1:
	UF : 1, UT : 1,		CONFIG : 'N U T, 0, 0, 1',
	X =  52.000  mm,	Y =  103.000  mm,	Z =   15.000 mm,
	W =180.000 deg,	P =   0.000 deg,	R =    90.000 deg
};
P[5521]{
   GP1:
	UF : 1, UT : 1,		CONFIG : 'N U T, 0, 0, 1',
	X =  58.000  mm,	Y =  103.000  mm,	Z =   15.000 mm,
	W =180.000 deg,	P =   0.000 deg,	R =    90.000 deg
};
P[5522]{
   GP1:
	UF : 1, UT : 1,		CONFIG : 'N U T, 0, 0, 1',
	X =  58.000  mm,	Y =  103.000  mm,	Z =   0.600 mm,
	W =180.000 deg,	P =   0.000 deg,	R =    90.000 deg
};
P[5523]{
   GP1:
	UF : 1, UT : 1,		CONFIG : 'N U T, 0, 0, 1',
	X =  58.000  mm,	Y =  103.000  mm,	Z =   15.000 mm,
	W =180.000 deg,	P =   0.000 deg,	R =    90.000 deg
};
P[5524]{
   GP1:
	UF : 1, UT : 1,		CONFIG : 'N U T, 0, 0, 1',
	X =  61.000  mm,	Y =  103.000  mm,	Z =   15.000 mm,
	W =180.000 deg,	P =   0.000 deg,	R =    90.000 deg
};
P[5525]{
   GP1:
	UF : 1, UT : 1,		CONFIG : 'N U T, 0, 0, 1',
	X =  61.000  mm,	Y =  103.000  mm,	Z =   0.600 mm,
	W =180.000 deg,	P =   0.000 deg,	R =    90.000 deg
};
P[5526]{
   GP1:
	UF : 1, UT : 1,		CONFIG : 'N U T, 0, 0, 1',
	X =  61.000  mm,	Y =  103.000  mm,	Z =   15.000 mm,
	W =180.000 deg,	P =   0.000 deg,	R =    90.000 deg
};
P[5527]{
   GP1:
	UF : 1, UT : 1,		CONFIG : 'N U T, 0, 0, 1',
	X =  64.000  mm,	Y =  103.000  mm,	Z =   15.000 mm,
	W =180.000 deg,	P =   0.000 deg,	R =    90.000 deg
};
P[5528]{
   GP1:
	UF : 1, UT : 1,		CONFIG : 'N U T, 0, 0, 1',
	X =  64.000  mm,	Y =  103.000  mm,	Z =   0.600 mm,
	W =180.000 deg,	P =   0.000 deg,	R =    90.000 deg
};
P[5529]{
   GP1:
	UF : 1, UT : 1,		CONFIG : 'N U T, 0, 0, 1',
	X =  64.000  mm,	Y =  103.000  mm,	Z =   15.000 mm,
	W =180.000 deg,	P =   0.000 deg,	R =    90.000 deg
};
P[5530]{
   GP1:
	UF : 1, UT : 1,		CONFIG : 'N U T, 0, 0, 1',
	X =  67.000  mm,	Y =  103.000  mm,	Z =   15.000 mm,
	W =180.000 deg,	P =   0.000 deg,	R =    90.000 deg
};
P[5531]{
   GP1:
	UF : 1, UT : 1,		CONFIG : 'N U T, 0, 0, 1',
	X =  67.000  mm,	Y =  103.000  mm,	Z =   0.600 mm,
	W =180.000 deg,	P =   0.000 deg,	R =    90.000 deg
};
P[5532]{
   GP1:
	UF : 1, UT : 1,		CONFIG : 'N U T, 0, 0, 1',
	X =  67.000  mm,	Y =  103.000  mm,	Z =   15.000 mm,
	W =180.000 deg,	P =   0.000 deg,	R =    90.000 deg
};
P[5533]{
   GP1:
	UF : 1, UT : 1,		CONFIG : 'N U T, 0, 0, 1',
	X =  70.000  mm,	Y =  103.000  mm,	Z =   15.000 mm,
	W =180.000 deg,	P =   0.000 deg,	R =    90.000 deg
};
P[5534]{
   GP1:
	UF : 1, UT : 1,		CONFIG : 'N U T, 0, 0, 1',
	X =  70.000  mm,	Y =  103.000  mm,	Z =   0.600 mm,
	W =180.000 deg,	P =   0.000 deg,	R =    90.000 deg
};
P[5535]{
   GP1:
	UF : 1, UT : 1,		CONFIG : 'N U T, 0, 0, 1',
	X =  70.000  mm,	Y =  103.000  mm,	Z =   15.000 mm,
	W =180.000 deg,	P =   0.000 deg,	R =    90.000 deg
};
P[5536]{
   GP1:
	UF : 1, UT : 1,		CONFIG : 'N U T, 0, 0, 1',
	X =  73.000  mm,	Y =  103.000  mm,	Z =   15.000 mm,
	W =180.000 deg,	P =   0.000 deg,	R =    90.000 deg
};
P[5537]{
   GP1:
	UF : 1, UT : 1,		CONFIG : 'N U T, 0, 0, 1',
	X =  73.000  mm,	Y =  103.000  mm,	Z =   0.600 mm,
	W =180.000 deg,	P =   0.000 deg,	R =    90.000 deg
};
P[5538]{
   GP1:
	UF : 1, UT : 1,		CONFIG : 'N U T, 0, 0, 1',
	X =  73.000  mm,	Y =  103.000  mm,	Z =   15.000 mm,
	W =180.000 deg,	P =   0.000 deg,	R =    90.000 deg
};
P[5539]{
   GP1:
	UF : 1, UT : 1,		CONFIG : 'N U T, 0, 0, 1',
	X =  76.000  mm,	Y =  103.000  mm,	Z =   15.000 mm,
	W =180.000 deg,	P =   0.000 deg,	R =    90.000 deg
};
P[5540]{
   GP1:
	UF : 1, UT : 1,		CONFIG : 'N U T, 0, 0, 1',
	X =  76.000  mm,	Y =  103.000  mm,	Z =   0.600 mm,
	W =180.000 deg,	P =   0.000 deg,	R =    90.000 deg
};
P[5541]{
   GP1:
	UF : 1, UT : 1,		CONFIG : 'N U T, 0, 0, 1',
	X =  76.000  mm,	Y =  103.000  mm,	Z =   15.000 mm,
	W =180.000 deg,	P =   0.000 deg,	R =    90.000 deg
};
P[5542]{
   GP1:
	UF : 1, UT : 1,		CONFIG : 'N U T, 0, 0, 1',
	X =  79.000  mm,	Y =  103.000  mm,	Z =   15.000 mm,
	W =180.000 deg,	P =   0.000 deg,	R =    90.000 deg
};
P[5543]{
   GP1:
	UF : 1, UT : 1,		CONFIG : 'N U T, 0, 0, 1',
	X =  79.000  mm,	Y =  103.000  mm,	Z =   0.600 mm,
	W =180.000 deg,	P =   0.000 deg,	R =    90.000 deg
};
P[5544]{
   GP1:
	UF : 1, UT : 1,		CONFIG : 'N U T, 0, 0, 1',
	X =  79.000  mm,	Y =  103.000  mm,	Z =   15.000 mm,
	W =180.000 deg,	P =   0.000 deg,	R =    90.000 deg
};
P[5545]{
   GP1:
	UF : 1, UT : 1,		CONFIG : 'N U T, 0, 0, 1',
	X =  82.000  mm,	Y =  103.000  mm,	Z =   15.000 mm,
	W =180.000 deg,	P =   0.000 deg,	R =    90.000 deg
};
P[5546]{
   GP1:
	UF : 1, UT : 1,		CONFIG : 'N U T, 0, 0, 1',
	X =  82.000  mm,	Y =  103.000  mm,	Z =   0.600 mm,
	W =180.000 deg,	P =   0.000 deg,	R =    90.000 deg
};
P[5547]{
   GP1:
	UF : 1, UT : 1,		CONFIG : 'N U T, 0, 0, 1',
	X =  82.000  mm,	Y =  103.000  mm,	Z =   15.000 mm,
	W =180.000 deg,	P =   0.000 deg,	R =    90.000 deg
};
P[5548]{
   GP1:
	UF : 1, UT : 1,		CONFIG : 'N U T, 0, 0, 1',
	X =  85.000  mm,	Y =  103.000  mm,	Z =   15.000 mm,
	W =180.000 deg,	P =   0.000 deg,	R =    90.000 deg
};
P[5549]{
   GP1:
	UF : 1, UT : 1,		CONFIG : 'N U T, 0, 0, 1',
	X =  85.000  mm,	Y =  103.000  mm,	Z =   0.600 mm,
	W =180.000 deg,	P =   0.000 deg,	R =    90.000 deg
};
P[5550]{
   GP1:
	UF : 1, UT : 1,		CONFIG : 'N U T, 0, 0, 1',
	X =  85.000  mm,	Y =  103.000  mm,	Z =   15.000 mm,
	W =180.000 deg,	P =   0.000 deg,	R =    90.000 deg
};
P[5551]{
   GP1:
	UF : 1, UT : 1,		CONFIG : 'N U T, 0, 0, 1',
	X =  88.000  mm,	Y =  103.000  mm,	Z =   15.000 mm,
	W =180.000 deg,	P =   0.000 deg,	R =    90.000 deg
};
P[5552]{
   GP1:
	UF : 1, UT : 1,		CONFIG : 'N U T, 0, 0, 1',
	X =  88.000  mm,	Y =  103.000  mm,	Z =   0.600 mm,
	W =180.000 deg,	P =   0.000 deg,	R =    90.000 deg
};
P[5553]{
   GP1:
	UF : 1, UT : 1,		CONFIG : 'N U T, 0, 0, 1',
	X =  88.000  mm,	Y =  103.000  mm,	Z =   15.000 mm,
	W =180.000 deg,	P =   0.000 deg,	R =    90.000 deg
};
P[5554]{
   GP1:
	UF : 1, UT : 1,		CONFIG : 'N U T, 0, 0, 1',
	X =  91.000  mm,	Y =  103.000  mm,	Z =   15.000 mm,
	W =180.000 deg,	P =   0.000 deg,	R =    90.000 deg
};
P[5555]{
   GP1:
	UF : 1, UT : 1,		CONFIG : 'N U T, 0, 0, 1',
	X =  91.000  mm,	Y =  103.000  mm,	Z =   0.600 mm,
	W =180.000 deg,	P =   0.000 deg,	R =    90.000 deg
};
P[5556]{
   GP1:
	UF : 1, UT : 1,		CONFIG : 'N U T, 0, 0, 1',
	X =  91.000  mm,	Y =  103.000  mm,	Z =   15.000 mm,
	W =180.000 deg,	P =   0.000 deg,	R =    90.000 deg
};
P[5557]{
   GP1:
	UF : 1, UT : 1,		CONFIG : 'N U T, 0, 0, 1',
	X =  94.000  mm,	Y =  103.000  mm,	Z =   15.000 mm,
	W =180.000 deg,	P =   0.000 deg,	R =    90.000 deg
};
P[5558]{
   GP1:
	UF : 1, UT : 1,		CONFIG : 'N U T, 0, 0, 1',
	X =  94.000  mm,	Y =  103.000  mm,	Z =   0.600 mm,
	W =180.000 deg,	P =   0.000 deg,	R =    90.000 deg
};
P[5559]{
   GP1:
	UF : 1, UT : 1,		CONFIG : 'N U T, 0, 0, 1',
	X =  94.000  mm,	Y =  103.000  mm,	Z =   15.000 mm,
	W =180.000 deg,	P =   0.000 deg,	R =    90.000 deg
};
P[5560]{
   GP1:
	UF : 1, UT : 1,		CONFIG : 'N U T, 0, 0, 1',
	X =  97.000  mm,	Y =  103.000  mm,	Z =   15.000 mm,
	W =180.000 deg,	P =   0.000 deg,	R =    90.000 deg
};
P[5561]{
   GP1:
	UF : 1, UT : 1,		CONFIG : 'N U T, 0, 0, 1',
	X =  97.000  mm,	Y =  103.000  mm,	Z =   0.600 mm,
	W =180.000 deg,	P =   0.000 deg,	R =    90.000 deg
};
P[5562]{
   GP1:
	UF : 1, UT : 1,		CONFIG : 'N U T, 0, 0, 1',
	X =  97.000  mm,	Y =  103.000  mm,	Z =   15.000 mm,
	W =180.000 deg,	P =   0.000 deg,	R =    90.000 deg
};
P[5563]{
   GP1:
	UF : 1, UT : 1,		CONFIG : 'N U T, 0, 0, 1',
	X =  100.000  mm,	Y =  103.000  mm,	Z =   15.000 mm,
	W =180.000 deg,	P =   0.000 deg,	R =    90.000 deg
};
P[5564]{
   GP1:
	UF : 1, UT : 1,		CONFIG : 'N U T, 0, 0, 1',
	X =  100.000  mm,	Y =  103.000  mm,	Z =   0.600 mm,
	W =180.000 deg,	P =   0.000 deg,	R =    90.000 deg
};
P[5565]{
   GP1:
	UF : 1, UT : 1,		CONFIG : 'N U T, 0, 0, 1',
	X =  100.000  mm,	Y =  103.000  mm,	Z =   15.000 mm,
	W =180.000 deg,	P =   0.000 deg,	R =    90.000 deg
};
P[5566]{
   GP1:
	UF : 1, UT : 1,		CONFIG : 'N U T, 0, 0, 1',
	X =  103.000  mm,	Y =  103.000  mm,	Z =   15.000 mm,
	W =180.000 deg,	P =   0.000 deg,	R =    90.000 deg
};
P[5567]{
   GP1:
	UF : 1, UT : 1,		CONFIG : 'N U T, 0, 0, 1',
	X =  103.000  mm,	Y =  103.000  mm,	Z =   0.600 mm,
	W =180.000 deg,	P =   0.000 deg,	R =    90.000 deg
};
P[5568]{
   GP1:
	UF : 1, UT : 1,		CONFIG : 'N U T, 0, 0, 1',
	X =  103.000  mm,	Y =  103.000  mm,	Z =   15.000 mm,
	W =180.000 deg,	P =   0.000 deg,	R =    90.000 deg
};
P[5569]{
   GP1:
	UF : 1, UT : 1,		CONFIG : 'N U T, 0, 0, 1',
	X =  106.000  mm,	Y =  103.000  mm,	Z =   15.000 mm,
	W =180.000 deg,	P =   0.000 deg,	R =    90.000 deg
};
P[5570]{
   GP1:
	UF : 1, UT : 1,		CONFIG : 'N U T, 0, 0, 1',
	X =  106.000  mm,	Y =  103.000  mm,	Z =   0.600 mm,
	W =180.000 deg,	P =   0.000 deg,	R =    90.000 deg
};
P[5571]{
   GP1:
	UF : 1, UT : 1,		CONFIG : 'N U T, 0, 0, 1',
	X =  106.000  mm,	Y =  103.000  mm,	Z =   15.000 mm,
	W =180.000 deg,	P =   0.000 deg,	R =    90.000 deg
};
P[5572]{
   GP1:
	UF : 1, UT : 1,		CONFIG : 'N U T, 0, 0, 1',
	X =  109.000  mm,	Y =  103.000  mm,	Z =   15.000 mm,
	W =180.000 deg,	P =   0.000 deg,	R =    90.000 deg
};
P[5573]{
   GP1:
	UF : 1, UT : 1,		CONFIG : 'N U T, 0, 0, 1',
	X =  109.000  mm,	Y =  103.000  mm,	Z =   0.600 mm,
	W =180.000 deg,	P =   0.000 deg,	R =    90.000 deg
};
P[5574]{
   GP1:
	UF : 1, UT : 1,		CONFIG : 'N U T, 0, 0, 1',
	X =  109.000  mm,	Y =  103.000  mm,	Z =   15.000 mm,
	W =180.000 deg,	P =   0.000 deg,	R =    90.000 deg
};
P[5575]{
   GP1:
	UF : 1, UT : 1,		CONFIG : 'N U T, 0, 0, 1',
	X =  112.000  mm,	Y =  103.000  mm,	Z =   15.000 mm,
	W =180.000 deg,	P =   0.000 deg,	R =    90.000 deg
};
P[5576]{
   GP1:
	UF : 1, UT : 1,		CONFIG : 'N U T, 0, 0, 1',
	X =  112.000  mm,	Y =  103.000  mm,	Z =   0.600 mm,
	W =180.000 deg,	P =   0.000 deg,	R =    90.000 deg
};
P[5577]{
   GP1:
	UF : 1, UT : 1,		CONFIG : 'N U T, 0, 0, 1',
	X =  112.000  mm,	Y =  103.000  mm,	Z =   15.000 mm,
	W =180.000 deg,	P =   0.000 deg,	R =    90.000 deg
};
P[5578]{
   GP1:
	UF : 1, UT : 1,		CONFIG : 'N U T, 0, 0, 1',
	X =  115.000  mm,	Y =  103.000  mm,	Z =   15.000 mm,
	W =180.000 deg,	P =   0.000 deg,	R =    90.000 deg
};
P[5579]{
   GP1:
	UF : 1, UT : 1,		CONFIG : 'N U T, 0, 0, 1',
	X =  115.000  mm,	Y =  103.000  mm,	Z =   0.600 mm,
	W =180.000 deg,	P =   0.000 deg,	R =    90.000 deg
};
P[5580]{
   GP1:
	UF : 1, UT : 1,		CONFIG : 'N U T, 0, 0, 1',
	X =  115.000  mm,	Y =  103.000  mm,	Z =   15.000 mm,
	W =180.000 deg,	P =   0.000 deg,	R =    90.000 deg
};
P[5581]{
   GP1:
	UF : 1, UT : 1,		CONFIG : 'N U T, 0, 0, 1',
	X =  118.000  mm,	Y =  103.000  mm,	Z =   15.000 mm,
	W =180.000 deg,	P =   0.000 deg,	R =    90.000 deg
};
P[5582]{
   GP1:
	UF : 1, UT : 1,		CONFIG : 'N U T, 0, 0, 1',
	X =  118.000  mm,	Y =  103.000  mm,	Z =   0.600 mm,
	W =180.000 deg,	P =   0.000 deg,	R =    90.000 deg
};
P[5583]{
   GP1:
	UF : 1, UT : 1,		CONFIG : 'N U T, 0, 0, 1',
	X =  118.000  mm,	Y =  103.000  mm,	Z =   15.000 mm,
	W =180.000 deg,	P =   0.000 deg,	R =    90.000 deg
};
P[5602]{
   GP1:
	UF : 1, UT : 1,		CONFIG : 'N U T, 0, 0, 1',
	X =  139.000  mm,	Y =  103.000  mm,	Z =   15.000 mm,
	W =180.000 deg,	P =   0.000 deg,	R =    90.000 deg
};
P[5603]{
   GP1:
	UF : 1, UT : 1,		CONFIG : 'N U T, 0, 0, 1',
	X =  139.000  mm,	Y =  103.000  mm,	Z =   0.600 mm,
	W =180.000 deg,	P =   0.000 deg,	R =    90.000 deg
};
P[5604]{
   GP1:
	UF : 1, UT : 1,		CONFIG : 'N U T, 0, 0, 1',
	X =  139.000  mm,	Y =  103.000  mm,	Z =   15.000 mm,
	W =180.000 deg,	P =   0.000 deg,	R =    90.000 deg
};
P[5605]{
   GP1:
	UF : 1, UT : 1,		CONFIG : 'N U T, 0, 0, 1',
	X =  142.000  mm,	Y =  103.000  mm,	Z =   15.000 mm,
	W =180.000 deg,	P =   0.000 deg,	R =    90.000 deg
};
P[5606]{
   GP1:
	UF : 1, UT : 1,		CONFIG : 'N U T, 0, 0, 1',
	X =  142.000  mm,	Y =  103.000  mm,	Z =   0.600 mm,
	W =180.000 deg,	P =   0.000 deg,	R =    90.000 deg
};
P[5607]{
   GP1:
	UF : 1, UT : 1,		CONFIG : 'N U T, 0, 0, 1',
	X =  142.000  mm,	Y =  103.000  mm,	Z =   15.000 mm,
	W =180.000 deg,	P =   0.000 deg,	R =    90.000 deg
};
P[5608]{
   GP1:
	UF : 1, UT : 1,		CONFIG : 'N U T, 0, 0, 1',
	X =  145.000  mm,	Y =  103.000  mm,	Z =   15.000 mm,
	W =180.000 deg,	P =   0.000 deg,	R =    90.000 deg
};
P[5609]{
   GP1:
	UF : 1, UT : 1,		CONFIG : 'N U T, 0, 0, 1',
	X =  145.000  mm,	Y =  103.000  mm,	Z =   0.600 mm,
	W =180.000 deg,	P =   0.000 deg,	R =    90.000 deg
};
P[5610]{
   GP1:
	UF : 1, UT : 1,		CONFIG : 'N U T, 0, 0, 1',
	X =  145.000  mm,	Y =  103.000  mm,	Z =   15.000 mm,
	W =180.000 deg,	P =   0.000 deg,	R =    90.000 deg
};
P[5617]{
   GP1:
	UF : 1, UT : 1,		CONFIG : 'N U T, 0, 0, 1',
	X =  163.000  mm,	Y =  103.000  mm,	Z =   15.000 mm,
	W =180.000 deg,	P =   0.000 deg,	R =    90.000 deg
};
P[5618]{
   GP1:
	UF : 1, UT : 1,		CONFIG : 'N U T, 0, 0, 1',
	X =  163.000  mm,	Y =  103.000  mm,	Z =   0.600 mm,
	W =180.000 deg,	P =   0.000 deg,	R =    90.000 deg
};
P[5619]{
   GP1:
	UF : 1, UT : 1,		CONFIG : 'N U T, 0, 0, 1',
	X =  163.000  mm,	Y =  103.000  mm,	Z =   15.000 mm,
	W =180.000 deg,	P =   0.000 deg,	R =    90.000 deg
};
P[5620]{
   GP1:
	UF : 1, UT : 1,		CONFIG : 'N U T, 0, 0, 1',
	X =  166.000  mm,	Y =  103.000  mm,	Z =   15.000 mm,
	W =180.000 deg,	P =   0.000 deg,	R =    90.000 deg
};
P[5621]{
   GP1:
	UF : 1, UT : 1,		CONFIG : 'N U T, 0, 0, 1',
	X =  166.000  mm,	Y =  103.000  mm,	Z =   0.600 mm,
	W =180.000 deg,	P =   0.000 deg,	R =    90.000 deg
};
P[5622]{
   GP1:
	UF : 1, UT : 1,		CONFIG : 'N U T, 0, 0, 1',
	X =  166.000  mm,	Y =  103.000  mm,	Z =   15.000 mm,
	W =180.000 deg,	P =   0.000 deg,	R =    90.000 deg
};
P[5623]{
   GP1:
	UF : 1, UT : 1,		CONFIG : 'N U T, 0, 0, 1',
	X =  169.000  mm,	Y =  103.000  mm,	Z =   15.000 mm,
	W =180.000 deg,	P =   0.000 deg,	R =    90.000 deg
};
P[5624]{
   GP1:
	UF : 1, UT : 1,		CONFIG : 'N U T, 0, 0, 1',
	X =  169.000  mm,	Y =  103.000  mm,	Z =   0.600 mm,
	W =180.000 deg,	P =   0.000 deg,	R =    90.000 deg
};
P[5625]{
   GP1:
	UF : 1, UT : 1,		CONFIG : 'N U T, 0, 0, 1',
	X =  169.000  mm,	Y =  103.000  mm,	Z =   15.000 mm,
	W =180.000 deg,	P =   0.000 deg,	R =    90.000 deg
};
P[5626]{
   GP1:
	UF : 1, UT : 1,		CONFIG : 'N U T, 0, 0, 1',
	X =  172.000  mm,	Y =  103.000  mm,	Z =   15.000 mm,
	W =180.000 deg,	P =   0.000 deg,	R =    90.000 deg
};
P[5627]{
   GP1:
	UF : 1, UT : 1,		CONFIG : 'N U T, 0, 0, 1',
	X =  172.000  mm,	Y =  103.000  mm,	Z =   0.600 mm,
	W =180.000 deg,	P =   0.000 deg,	R =    90.000 deg
};
P[5628]{
   GP1:
	UF : 1, UT : 1,		CONFIG : 'N U T, 0, 0, 1',
	X =  172.000  mm,	Y =  103.000  mm,	Z =   15.000 mm,
	W =180.000 deg,	P =   0.000 deg,	R =    90.000 deg
};
P[5629]{
   GP1:
	UF : 1, UT : 1,		CONFIG : 'N U T, 0, 0, 1',
	X =  175.000  mm,	Y =  103.000  mm,	Z =   15.000 mm,
	W =180.000 deg,	P =   0.000 deg,	R =    90.000 deg
};
P[5630]{
   GP1:
	UF : 1, UT : 1,		CONFIG : 'N U T, 0, 0, 1',
	X =  175.000  mm,	Y =  103.000  mm,	Z =   0.600 mm,
	W =180.000 deg,	P =   0.000 deg,	R =    90.000 deg
};
P[5631]{
   GP1:
	UF : 1, UT : 1,		CONFIG : 'N U T, 0, 0, 1',
	X =  175.000  mm,	Y =  103.000  mm,	Z =   15.000 mm,
	W =180.000 deg,	P =   0.000 deg,	R =    90.000 deg
};
P[5632]{
   GP1:
	UF : 1, UT : 1,		CONFIG : 'N U T, 0, 0, 1',
	X =  178.000  mm,	Y =  103.000  mm,	Z =   15.000 mm,
	W =180.000 deg,	P =   0.000 deg,	R =    90.000 deg
};
P[5633]{
   GP1:
	UF : 1, UT : 1,		CONFIG : 'N U T, 0, 0, 1',
	X =  178.000  mm,	Y =  103.000  mm,	Z =   0.600 mm,
	W =180.000 deg,	P =   0.000 deg,	R =    90.000 deg
};
P[5634]{
   GP1:
	UF : 1, UT : 1,		CONFIG : 'N U T, 0, 0, 1',
	X =  178.000  mm,	Y =  103.000  mm,	Z =   15.000 mm,
	W =180.000 deg,	P =   0.000 deg,	R =    90.000 deg
};
P[5641]{
   GP1:
	UF : 1, UT : 1,		CONFIG : 'N U T, 0, 0, 1',
	X =  7.000  mm,	Y =  106.000  mm,	Z =   15.000 mm,
	W =180.000 deg,	P =   0.000 deg,	R =    90.000 deg
};
P[5642]{
   GP1:
	UF : 1, UT : 1,		CONFIG : 'N U T, 0, 0, 1',
	X =  7.000  mm,	Y =  106.000  mm,	Z =   0.600 mm,
	W =180.000 deg,	P =   0.000 deg,	R =    90.000 deg
};
P[5643]{
   GP1:
	UF : 1, UT : 1,		CONFIG : 'N U T, 0, 0, 1',
	X =  7.000  mm,	Y =  106.000  mm,	Z =   15.000 mm,
	W =180.000 deg,	P =   0.000 deg,	R =    90.000 deg
};
P[5644]{
   GP1:
	UF : 1, UT : 1,		CONFIG : 'N U T, 0, 0, 1',
	X =  10.000  mm,	Y =  106.000  mm,	Z =   15.000 mm,
	W =180.000 deg,	P =   0.000 deg,	R =    90.000 deg
};
P[5645]{
   GP1:
	UF : 1, UT : 1,		CONFIG : 'N U T, 0, 0, 1',
	X =  10.000  mm,	Y =  106.000  mm,	Z =   0.600 mm,
	W =180.000 deg,	P =   0.000 deg,	R =    90.000 deg
};
P[5646]{
   GP1:
	UF : 1, UT : 1,		CONFIG : 'N U T, 0, 0, 1',
	X =  10.000  mm,	Y =  106.000  mm,	Z =   15.000 mm,
	W =180.000 deg,	P =   0.000 deg,	R =    90.000 deg
};
P[5647]{
   GP1:
	UF : 1, UT : 1,		CONFIG : 'N U T, 0, 0, 1',
	X =  13.000  mm,	Y =  106.000  mm,	Z =   15.000 mm,
	W =180.000 deg,	P =   0.000 deg,	R =    90.000 deg
};
P[5648]{
   GP1:
	UF : 1, UT : 1,		CONFIG : 'N U T, 0, 0, 1',
	X =  13.000  mm,	Y =  106.000  mm,	Z =   0.600 mm,
	W =180.000 deg,	P =   0.000 deg,	R =    90.000 deg
};
P[5649]{
   GP1:
	UF : 1, UT : 1,		CONFIG : 'N U T, 0, 0, 1',
	X =  13.000  mm,	Y =  106.000  mm,	Z =   15.000 mm,
	W =180.000 deg,	P =   0.000 deg,	R =    90.000 deg
};
P[5650]{
   GP1:
	UF : 1, UT : 1,		CONFIG : 'N U T, 0, 0, 1',
	X =  16.000  mm,	Y =  106.000  mm,	Z =   15.000 mm,
	W =180.000 deg,	P =   0.000 deg,	R =    90.000 deg
};
P[5651]{
   GP1:
	UF : 1, UT : 1,		CONFIG : 'N U T, 0, 0, 1',
	X =  16.000  mm,	Y =  106.000  mm,	Z =   0.600 mm,
	W =180.000 deg,	P =   0.000 deg,	R =    90.000 deg
};
P[5652]{
   GP1:
	UF : 1, UT : 1,		CONFIG : 'N U T, 0, 0, 1',
	X =  16.000  mm,	Y =  106.000  mm,	Z =   15.000 mm,
	W =180.000 deg,	P =   0.000 deg,	R =    90.000 deg
};
P[5668]{
   GP1:
	UF : 1, UT : 1,		CONFIG : 'N U T, 0, 0, 1',
	X =  34.000  mm,	Y =  106.000  mm,	Z =   15.000 mm,
	W =180.000 deg,	P =   0.000 deg,	R =    90.000 deg
};
P[5669]{
   GP1:
	UF : 1, UT : 1,		CONFIG : 'N U T, 0, 0, 1',
	X =  34.000  mm,	Y =  106.000  mm,	Z =   0.600 mm,
	W =180.000 deg,	P =   0.000 deg,	R =    90.000 deg
};
P[5670]{
   GP1:
	UF : 1, UT : 1,		CONFIG : 'N U T, 0, 0, 1',
	X =  34.000  mm,	Y =  106.000  mm,	Z =   15.000 mm,
	W =180.000 deg,	P =   0.000 deg,	R =    90.000 deg
};
P[5671]{
   GP1:
	UF : 1, UT : 1,		CONFIG : 'N U T, 0, 0, 1',
	X =  37.000  mm,	Y =  106.000  mm,	Z =   15.000 mm,
	W =180.000 deg,	P =   0.000 deg,	R =    90.000 deg
};
P[5672]{
   GP1:
	UF : 1, UT : 1,		CONFIG : 'N U T, 0, 0, 1',
	X =  37.000  mm,	Y =  106.000  mm,	Z =   0.600 mm,
	W =180.000 deg,	P =   0.000 deg,	R =    90.000 deg
};
P[5673]{
   GP1:
	UF : 1, UT : 1,		CONFIG : 'N U T, 0, 0, 1',
	X =  37.000  mm,	Y =  106.000  mm,	Z =   15.000 mm,
	W =180.000 deg,	P =   0.000 deg,	R =    90.000 deg
};
P[5674]{
   GP1:
	UF : 1, UT : 1,		CONFIG : 'N U T, 0, 0, 1',
	X =  40.000  mm,	Y =  106.000  mm,	Z =   15.000 mm,
	W =180.000 deg,	P =   0.000 deg,	R =    90.000 deg
};
P[5675]{
   GP1:
	UF : 1, UT : 1,		CONFIG : 'N U T, 0, 0, 1',
	X =  40.000  mm,	Y =  106.000  mm,	Z =   0.600 mm,
	W =180.000 deg,	P =   0.000 deg,	R =    90.000 deg
};
P[5676]{
   GP1:
	UF : 1, UT : 1,		CONFIG : 'N U T, 0, 0, 1',
	X =  40.000  mm,	Y =  106.000  mm,	Z =   15.000 mm,
	W =180.000 deg,	P =   0.000 deg,	R =    90.000 deg
};
P[5680]{
   GP1:
	UF : 1, UT : 1,		CONFIG : 'N U T, 0, 0, 1',
	X =  46.000  mm,	Y =  106.000  mm,	Z =   15.000 mm,
	W =180.000 deg,	P =   0.000 deg,	R =    90.000 deg
};
P[5681]{
   GP1:
	UF : 1, UT : 1,		CONFIG : 'N U T, 0, 0, 1',
	X =  46.000  mm,	Y =  106.000  mm,	Z =   0.600 mm,
	W =180.000 deg,	P =   0.000 deg,	R =    90.000 deg
};
P[5682]{
   GP1:
	UF : 1, UT : 1,		CONFIG : 'N U T, 0, 0, 1',
	X =  46.000  mm,	Y =  106.000  mm,	Z =   15.000 mm,
	W =180.000 deg,	P =   0.000 deg,	R =    90.000 deg
};
P[5683]{
   GP1:
	UF : 1, UT : 1,		CONFIG : 'N U T, 0, 0, 1',
	X =  49.000  mm,	Y =  106.000  mm,	Z =   15.000 mm,
	W =180.000 deg,	P =   0.000 deg,	R =    90.000 deg
};
P[5684]{
   GP1:
	UF : 1, UT : 1,		CONFIG : 'N U T, 0, 0, 1',
	X =  49.000  mm,	Y =  106.000  mm,	Z =   0.600 mm,
	W =180.000 deg,	P =   0.000 deg,	R =    90.000 deg
};
P[5685]{
   GP1:
	UF : 1, UT : 1,		CONFIG : 'N U T, 0, 0, 1',
	X =  49.000  mm,	Y =  106.000  mm,	Z =   15.000 mm,
	W =180.000 deg,	P =   0.000 deg,	R =    90.000 deg
};
P[5686]{
   GP1:
	UF : 1, UT : 1,		CONFIG : 'N U T, 0, 0, 1',
	X =  52.000  mm,	Y =  106.000  mm,	Z =   15.000 mm,
	W =180.000 deg,	P =   0.000 deg,	R =    90.000 deg
};
P[5687]{
   GP1:
	UF : 1, UT : 1,		CONFIG : 'N U T, 0, 0, 1',
	X =  52.000  mm,	Y =  106.000  mm,	Z =   0.600 mm,
	W =180.000 deg,	P =   0.000 deg,	R =    90.000 deg
};
P[5688]{
   GP1:
	UF : 1, UT : 1,		CONFIG : 'N U T, 0, 0, 1',
	X =  52.000  mm,	Y =  106.000  mm,	Z =   15.000 mm,
	W =180.000 deg,	P =   0.000 deg,	R =    90.000 deg
};
P[5695]{
   GP1:
	UF : 1, UT : 1,		CONFIG : 'N U T, 0, 0, 1',
	X =  103.000  mm,	Y =  106.000  mm,	Z =   15.000 mm,
	W =180.000 deg,	P =   0.000 deg,	R =    90.000 deg
};
P[5696]{
   GP1:
	UF : 1, UT : 1,		CONFIG : 'N U T, 0, 0, 1',
	X =  103.000  mm,	Y =  106.000  mm,	Z =   0.600 mm,
	W =180.000 deg,	P =   0.000 deg,	R =    90.000 deg
};
P[5697]{
   GP1:
	UF : 1, UT : 1,		CONFIG : 'N U T, 0, 0, 1',
	X =  103.000  mm,	Y =  106.000  mm,	Z =   15.000 mm,
	W =180.000 deg,	P =   0.000 deg,	R =    90.000 deg
};
P[5698]{
   GP1:
	UF : 1, UT : 1,		CONFIG : 'N U T, 0, 0, 1',
	X =  106.000  mm,	Y =  106.000  mm,	Z =   15.000 mm,
	W =180.000 deg,	P =   0.000 deg,	R =    90.000 deg
};
P[5699]{
   GP1:
	UF : 1, UT : 1,		CONFIG : 'N U T, 0, 0, 1',
	X =  106.000  mm,	Y =  106.000  mm,	Z =   0.600 mm,
	W =180.000 deg,	P =   0.000 deg,	R =    90.000 deg
};
P[5700]{
   GP1:
	UF : 1, UT : 1,		CONFIG : 'N U T, 0, 0, 1',
	X =  106.000  mm,	Y =  106.000  mm,	Z =   15.000 mm,
	W =180.000 deg,	P =   0.000 deg,	R =    90.000 deg
};
P[5701]{
   GP1:
	UF : 1, UT : 1,		CONFIG : 'N U T, 0, 0, 1',
	X =  109.000  mm,	Y =  106.000  mm,	Z =   15.000 mm,
	W =180.000 deg,	P =   0.000 deg,	R =    90.000 deg
};
P[5702]{
   GP1:
	UF : 1, UT : 1,		CONFIG : 'N U T, 0, 0, 1',
	X =  109.000  mm,	Y =  106.000  mm,	Z =   0.600 mm,
	W =180.000 deg,	P =   0.000 deg,	R =    90.000 deg
};
P[5703]{
   GP1:
	UF : 1, UT : 1,		CONFIG : 'N U T, 0, 0, 1',
	X =  109.000  mm,	Y =  106.000  mm,	Z =   15.000 mm,
	W =180.000 deg,	P =   0.000 deg,	R =    90.000 deg
};
P[5704]{
   GP1:
	UF : 1, UT : 1,		CONFIG : 'N U T, 0, 0, 1',
	X =  112.000  mm,	Y =  106.000  mm,	Z =   15.000 mm,
	W =180.000 deg,	P =   0.000 deg,	R =    90.000 deg
};
P[5705]{
   GP1:
	UF : 1, UT : 1,		CONFIG : 'N U T, 0, 0, 1',
	X =  112.000  mm,	Y =  106.000  mm,	Z =   0.600 mm,
	W =180.000 deg,	P =   0.000 deg,	R =    90.000 deg
};
P[5706]{
   GP1:
	UF : 1, UT : 1,		CONFIG : 'N U T, 0, 0, 1',
	X =  112.000  mm,	Y =  106.000  mm,	Z =   15.000 mm,
	W =180.000 deg,	P =   0.000 deg,	R =    90.000 deg
};
P[5707]{
   GP1:
	UF : 1, UT : 1,		CONFIG : 'N U T, 0, 0, 1',
	X =  115.000  mm,	Y =  106.000  mm,	Z =   15.000 mm,
	W =180.000 deg,	P =   0.000 deg,	R =    90.000 deg
};
P[5708]{
   GP1:
	UF : 1, UT : 1,		CONFIG : 'N U T, 0, 0, 1',
	X =  115.000  mm,	Y =  106.000  mm,	Z =   0.600 mm,
	W =180.000 deg,	P =   0.000 deg,	R =    90.000 deg
};
P[5709]{
   GP1:
	UF : 1, UT : 1,		CONFIG : 'N U T, 0, 0, 1',
	X =  115.000  mm,	Y =  106.000  mm,	Z =   15.000 mm,
	W =180.000 deg,	P =   0.000 deg,	R =    90.000 deg
};
P[5710]{
   GP1:
	UF : 1, UT : 1,		CONFIG : 'N U T, 0, 0, 1',
	X =  118.000  mm,	Y =  106.000  mm,	Z =   15.000 mm,
	W =180.000 deg,	P =   0.000 deg,	R =    90.000 deg
};
P[5711]{
   GP1:
	UF : 1, UT : 1,		CONFIG : 'N U T, 0, 0, 1',
	X =  118.000  mm,	Y =  106.000  mm,	Z =   0.600 mm,
	W =180.000 deg,	P =   0.000 deg,	R =    90.000 deg
};
P[5712]{
   GP1:
	UF : 1, UT : 1,		CONFIG : 'N U T, 0, 0, 1',
	X =  118.000  mm,	Y =  106.000  mm,	Z =   15.000 mm,
	W =180.000 deg,	P =   0.000 deg,	R =    90.000 deg
};
P[5725]{
   GP1:
	UF : 1, UT : 1,		CONFIG : 'N U T, 0, 0, 1',
	X =  133.000  mm,	Y =  106.000  mm,	Z =   15.000 mm,
	W =180.000 deg,	P =   0.000 deg,	R =    90.000 deg
};
P[5726]{
   GP1:
	UF : 1, UT : 1,		CONFIG : 'N U T, 0, 0, 1',
	X =  133.000  mm,	Y =  106.000  mm,	Z =   0.600 mm,
	W =180.000 deg,	P =   0.000 deg,	R =    90.000 deg
};
P[5727]{
   GP1:
	UF : 1, UT : 1,		CONFIG : 'N U T, 0, 0, 1',
	X =  133.000  mm,	Y =  106.000  mm,	Z =   15.000 mm,
	W =180.000 deg,	P =   0.000 deg,	R =    90.000 deg
};
P[5728]{
   GP1:
	UF : 1, UT : 1,		CONFIG : 'N U T, 0, 0, 1',
	X =  136.000  mm,	Y =  106.000  mm,	Z =   15.000 mm,
	W =180.000 deg,	P =   0.000 deg,	R =    90.000 deg
};
P[5729]{
   GP1:
	UF : 1, UT : 1,		CONFIG : 'N U T, 0, 0, 1',
	X =  136.000  mm,	Y =  106.000  mm,	Z =   0.600 mm,
	W =180.000 deg,	P =   0.000 deg,	R =    90.000 deg
};
P[5730]{
   GP1:
	UF : 1, UT : 1,		CONFIG : 'N U T, 0, 0, 1',
	X =  136.000  mm,	Y =  106.000  mm,	Z =   15.000 mm,
	W =180.000 deg,	P =   0.000 deg,	R =    90.000 deg
};
P[5731]{
   GP1:
	UF : 1, UT : 1,		CONFIG : 'N U T, 0, 0, 1',
	X =  139.000  mm,	Y =  106.000  mm,	Z =   15.000 mm,
	W =180.000 deg,	P =   0.000 deg,	R =    90.000 deg
};
P[5732]{
   GP1:
	UF : 1, UT : 1,		CONFIG : 'N U T, 0, 0, 1',
	X =  139.000  mm,	Y =  106.000  mm,	Z =   0.600 mm,
	W =180.000 deg,	P =   0.000 deg,	R =    90.000 deg
};
P[5733]{
   GP1:
	UF : 1, UT : 1,		CONFIG : 'N U T, 0, 0, 1',
	X =  139.000  mm,	Y =  106.000  mm,	Z =   15.000 mm,
	W =180.000 deg,	P =   0.000 deg,	R =    90.000 deg
};
P[5737]{
   GP1:
	UF : 1, UT : 1,		CONFIG : 'N U T, 0, 0, 1',
	X =  145.000  mm,	Y =  106.000  mm,	Z =   15.000 mm,
	W =180.000 deg,	P =   0.000 deg,	R =    90.000 deg
};
P[5738]{
   GP1:
	UF : 1, UT : 1,		CONFIG : 'N U T, 0, 0, 1',
	X =  145.000  mm,	Y =  106.000  mm,	Z =   0.600 mm,
	W =180.000 deg,	P =   0.000 deg,	R =    90.000 deg
};
P[5739]{
   GP1:
	UF : 1, UT : 1,		CONFIG : 'N U T, 0, 0, 1',
	X =  145.000  mm,	Y =  106.000  mm,	Z =   15.000 mm,
	W =180.000 deg,	P =   0.000 deg,	R =    90.000 deg
};
P[5743]{
   GP1:
	UF : 1, UT : 1,		CONFIG : 'N U T, 0, 0, 1',
	X =  163.000  mm,	Y =  106.000  mm,	Z =   15.000 mm,
	W =180.000 deg,	P =   0.000 deg,	R =    90.000 deg
};
P[5744]{
   GP1:
	UF : 1, UT : 1,		CONFIG : 'N U T, 0, 0, 1',
	X =  163.000  mm,	Y =  106.000  mm,	Z =   0.600 mm,
	W =180.000 deg,	P =   0.000 deg,	R =    90.000 deg
};
P[5745]{
   GP1:
	UF : 1, UT : 1,		CONFIG : 'N U T, 0, 0, 1',
	X =  163.000  mm,	Y =  106.000  mm,	Z =   15.000 mm,
	W =180.000 deg,	P =   0.000 deg,	R =    90.000 deg
};
P[5746]{
   GP1:
	UF : 1, UT : 1,		CONFIG : 'N U T, 0, 0, 1',
	X =  166.000  mm,	Y =  106.000  mm,	Z =   15.000 mm,
	W =180.000 deg,	P =   0.000 deg,	R =    90.000 deg
};
P[5747]{
   GP1:
	UF : 1, UT : 1,		CONFIG : 'N U T, 0, 0, 1',
	X =  166.000  mm,	Y =  106.000  mm,	Z =   0.600 mm,
	W =180.000 deg,	P =   0.000 deg,	R =    90.000 deg
};
P[5748]{
   GP1:
	UF : 1, UT : 1,		CONFIG : 'N U T, 0, 0, 1',
	X =  166.000  mm,	Y =  106.000  mm,	Z =   15.000 mm,
	W =180.000 deg,	P =   0.000 deg,	R =    90.000 deg
};
P[5749]{
   GP1:
	UF : 1, UT : 1,		CONFIG : 'N U T, 0, 0, 1',
	X =  169.000  mm,	Y =  106.000  mm,	Z =   15.000 mm,
	W =180.000 deg,	P =   0.000 deg,	R =    90.000 deg
};
P[5750]{
   GP1:
	UF : 1, UT : 1,		CONFIG : 'N U T, 0, 0, 1',
	X =  169.000  mm,	Y =  106.000  mm,	Z =   0.600 mm,
	W =180.000 deg,	P =   0.000 deg,	R =    90.000 deg
};
P[5751]{
   GP1:
	UF : 1, UT : 1,		CONFIG : 'N U T, 0, 0, 1',
	X =  169.000  mm,	Y =  106.000  mm,	Z =   15.000 mm,
	W =180.000 deg,	P =   0.000 deg,	R =    90.000 deg
};
P[5752]{
   GP1:
	UF : 1, UT : 1,		CONFIG : 'N U T, 0, 0, 1',
	X =  172.000  mm,	Y =  106.000  mm,	Z =   15.000 mm,
	W =180.000 deg,	P =   0.000 deg,	R =    90.000 deg
};
P[5753]{
   GP1:
	UF : 1, UT : 1,		CONFIG : 'N U T, 0, 0, 1',
	X =  172.000  mm,	Y =  106.000  mm,	Z =   0.600 mm,
	W =180.000 deg,	P =   0.000 deg,	R =    90.000 deg
};
P[5754]{
   GP1:
	UF : 1, UT : 1,		CONFIG : 'N U T, 0, 0, 1',
	X =  172.000  mm,	Y =  106.000  mm,	Z =   15.000 mm,
	W =180.000 deg,	P =   0.000 deg,	R =    90.000 deg
};
P[5755]{
   GP1:
	UF : 1, UT : 1,		CONFIG : 'N U T, 0, 0, 1',
	X =  175.000  mm,	Y =  106.000  mm,	Z =   15.000 mm,
	W =180.000 deg,	P =   0.000 deg,	R =    90.000 deg
};
P[5756]{
   GP1:
	UF : 1, UT : 1,		CONFIG : 'N U T, 0, 0, 1',
	X =  175.000  mm,	Y =  106.000  mm,	Z =   0.600 mm,
	W =180.000 deg,	P =   0.000 deg,	R =    90.000 deg
};
P[5757]{
   GP1:
	UF : 1, UT : 1,		CONFIG : 'N U T, 0, 0, 1',
	X =  175.000  mm,	Y =  106.000  mm,	Z =   15.000 mm,
	W =180.000 deg,	P =   0.000 deg,	R =    90.000 deg
};
P[5758]{
   GP1:
	UF : 1, UT : 1,		CONFIG : 'N U T, 0, 0, 1',
	X =  178.000  mm,	Y =  106.000  mm,	Z =   15.000 mm,
	W =180.000 deg,	P =   0.000 deg,	R =    90.000 deg
};
P[5759]{
   GP1:
	UF : 1, UT : 1,		CONFIG : 'N U T, 0, 0, 1',
	X =  178.000  mm,	Y =  106.000  mm,	Z =   0.600 mm,
	W =180.000 deg,	P =   0.000 deg,	R =    90.000 deg
};
P[5760]{
   GP1:
	UF : 1, UT : 1,		CONFIG : 'N U T, 0, 0, 1',
	X =  178.000  mm,	Y =  106.000  mm,	Z =   15.000 mm,
	W =180.000 deg,	P =   0.000 deg,	R =    90.000 deg
};
P[5761]{
   GP1:
	UF : 1, UT : 1,		CONFIG : 'N U T, 0, 0, 1',
	X =  1.000  mm,	Y =  109.000  mm,	Z =   15.000 mm,
	W =180.000 deg,	P =   0.000 deg,	R =    90.000 deg
};
P[5762]{
   GP1:
	UF : 1, UT : 1,		CONFIG : 'N U T, 0, 0, 1',
	X =  1.000  mm,	Y =  109.000  mm,	Z =   0.600 mm,
	W =180.000 deg,	P =   0.000 deg,	R =    90.000 deg
};
P[5763]{
   GP1:
	UF : 1, UT : 1,		CONFIG : 'N U T, 0, 0, 1',
	X =  1.000  mm,	Y =  109.000  mm,	Z =   15.000 mm,
	W =180.000 deg,	P =   0.000 deg,	R =    90.000 deg
};
P[5767]{
   GP1:
	UF : 1, UT : 1,		CONFIG : 'N U T, 0, 0, 1',
	X =  10.000  mm,	Y =  109.000  mm,	Z =   15.000 mm,
	W =180.000 deg,	P =   0.000 deg,	R =    90.000 deg
};
P[5768]{
   GP1:
	UF : 1, UT : 1,		CONFIG : 'N U T, 0, 0, 1',
	X =  10.000  mm,	Y =  109.000  mm,	Z =   0.600 mm,
	W =180.000 deg,	P =   0.000 deg,	R =    90.000 deg
};
P[5769]{
   GP1:
	UF : 1, UT : 1,		CONFIG : 'N U T, 0, 0, 1',
	X =  10.000  mm,	Y =  109.000  mm,	Z =   15.000 mm,
	W =180.000 deg,	P =   0.000 deg,	R =    90.000 deg
};
P[5770]{
   GP1:
	UF : 1, UT : 1,		CONFIG : 'N U T, 0, 0, 1',
	X =  13.000  mm,	Y =  109.000  mm,	Z =   15.000 mm,
	W =180.000 deg,	P =   0.000 deg,	R =    90.000 deg
};
P[5771]{
   GP1:
	UF : 1, UT : 1,		CONFIG : 'N U T, 0, 0, 1',
	X =  13.000  mm,	Y =  109.000  mm,	Z =   0.600 mm,
	W =180.000 deg,	P =   0.000 deg,	R =    90.000 deg
};
P[5772]{
   GP1:
	UF : 1, UT : 1,		CONFIG : 'N U T, 0, 0, 1',
	X =  13.000  mm,	Y =  109.000  mm,	Z =   15.000 mm,
	W =180.000 deg,	P =   0.000 deg,	R =    90.000 deg
};
P[5773]{
   GP1:
	UF : 1, UT : 1,		CONFIG : 'N U T, 0, 0, 1',
	X =  16.000  mm,	Y =  109.000  mm,	Z =   15.000 mm,
	W =180.000 deg,	P =   0.000 deg,	R =    90.000 deg
};
P[5774]{
   GP1:
	UF : 1, UT : 1,		CONFIG : 'N U T, 0, 0, 1',
	X =  16.000  mm,	Y =  109.000  mm,	Z =   0.600 mm,
	W =180.000 deg,	P =   0.000 deg,	R =    90.000 deg
};
P[5775]{
   GP1:
	UF : 1, UT : 1,		CONFIG : 'N U T, 0, 0, 1',
	X =  16.000  mm,	Y =  109.000  mm,	Z =   15.000 mm,
	W =180.000 deg,	P =   0.000 deg,	R =    90.000 deg
};
P[5776]{
   GP1:
	UF : 1, UT : 1,		CONFIG : 'N U T, 0, 0, 1',
	X =  19.000  mm,	Y =  109.000  mm,	Z =   15.000 mm,
	W =180.000 deg,	P =   0.000 deg,	R =    90.000 deg
};
P[5777]{
   GP1:
	UF : 1, UT : 1,		CONFIG : 'N U T, 0, 0, 1',
	X =  19.000  mm,	Y =  109.000  mm,	Z =   0.600 mm,
	W =180.000 deg,	P =   0.000 deg,	R =    90.000 deg
};
P[5778]{
   GP1:
	UF : 1, UT : 1,		CONFIG : 'N U T, 0, 0, 1',
	X =  19.000  mm,	Y =  109.000  mm,	Z =   15.000 mm,
	W =180.000 deg,	P =   0.000 deg,	R =    90.000 deg
};
P[5788]{
   GP1:
	UF : 1, UT : 1,		CONFIG : 'N U T, 0, 0, 1',
	X =  31.000  mm,	Y =  109.000  mm,	Z =   15.000 mm,
	W =180.000 deg,	P =   0.000 deg,	R =    90.000 deg
};
P[5789]{
   GP1:
	UF : 1, UT : 1,		CONFIG : 'N U T, 0, 0, 1',
	X =  31.000  mm,	Y =  109.000  mm,	Z =   0.600 mm,
	W =180.000 deg,	P =   0.000 deg,	R =    90.000 deg
};
P[5790]{
   GP1:
	UF : 1, UT : 1,		CONFIG : 'N U T, 0, 0, 1',
	X =  31.000  mm,	Y =  109.000  mm,	Z =   15.000 mm,
	W =180.000 deg,	P =   0.000 deg,	R =    90.000 deg
};
P[5806]{
   GP1:
	UF : 1, UT : 1,		CONFIG : 'N U T, 0, 0, 1',
	X =  49.000  mm,	Y =  109.000  mm,	Z =   15.000 mm,
	W =180.000 deg,	P =   0.000 deg,	R =    90.000 deg
};
P[5807]{
   GP1:
	UF : 1, UT : 1,		CONFIG : 'N U T, 0, 0, 1',
	X =  49.000  mm,	Y =  109.000  mm,	Z =   0.600 mm,
	W =180.000 deg,	P =   0.000 deg,	R =    90.000 deg
};
P[5808]{
   GP1:
	UF : 1, UT : 1,		CONFIG : 'N U T, 0, 0, 1',
	X =  49.000  mm,	Y =  109.000  mm,	Z =   15.000 mm,
	W =180.000 deg,	P =   0.000 deg,	R =    90.000 deg
};
P[5809]{
   GP1:
	UF : 1, UT : 1,		CONFIG : 'N U T, 0, 0, 1',
	X =  52.000  mm,	Y =  109.000  mm,	Z =   15.000 mm,
	W =180.000 deg,	P =   0.000 deg,	R =    90.000 deg
};
P[5810]{
   GP1:
	UF : 1, UT : 1,		CONFIG : 'N U T, 0, 0, 1',
	X =  52.000  mm,	Y =  109.000  mm,	Z =   0.600 mm,
	W =180.000 deg,	P =   0.000 deg,	R =    90.000 deg
};
P[5811]{
   GP1:
	UF : 1, UT : 1,		CONFIG : 'N U T, 0, 0, 1',
	X =  52.000  mm,	Y =  109.000  mm,	Z =   15.000 mm,
	W =180.000 deg,	P =   0.000 deg,	R =    90.000 deg
};
P[5815]{
   GP1:
	UF : 1, UT : 1,		CONFIG : 'N U T, 0, 0, 1',
	X =  109.000  mm,	Y =  109.000  mm,	Z =   15.000 mm,
	W =180.000 deg,	P =   0.000 deg,	R =    90.000 deg
};
P[5816]{
   GP1:
	UF : 1, UT : 1,		CONFIG : 'N U T, 0, 0, 1',
	X =  109.000  mm,	Y =  109.000  mm,	Z =   0.600 mm,
	W =180.000 deg,	P =   0.000 deg,	R =    90.000 deg
};
P[5817]{
   GP1:
	UF : 1, UT : 1,		CONFIG : 'N U T, 0, 0, 1',
	X =  109.000  mm,	Y =  109.000  mm,	Z =   15.000 mm,
	W =180.000 deg,	P =   0.000 deg,	R =    90.000 deg
};
P[5818]{
   GP1:
	UF : 1, UT : 1,		CONFIG : 'N U T, 0, 0, 1',
	X =  112.000  mm,	Y =  109.000  mm,	Z =   15.000 mm,
	W =180.000 deg,	P =   0.000 deg,	R =    90.000 deg
};
P[5819]{
   GP1:
	UF : 1, UT : 1,		CONFIG : 'N U T, 0, 0, 1',
	X =  112.000  mm,	Y =  109.000  mm,	Z =   0.600 mm,
	W =180.000 deg,	P =   0.000 deg,	R =    90.000 deg
};
P[5820]{
   GP1:
	UF : 1, UT : 1,		CONFIG : 'N U T, 0, 0, 1',
	X =  112.000  mm,	Y =  109.000  mm,	Z =   15.000 mm,
	W =180.000 deg,	P =   0.000 deg,	R =    90.000 deg
};
P[5821]{
   GP1:
	UF : 1, UT : 1,		CONFIG : 'N U T, 0, 0, 1',
	X =  115.000  mm,	Y =  109.000  mm,	Z =   15.000 mm,
	W =180.000 deg,	P =   0.000 deg,	R =    90.000 deg
};
P[5822]{
   GP1:
	UF : 1, UT : 1,		CONFIG : 'N U T, 0, 0, 1',
	X =  115.000  mm,	Y =  109.000  mm,	Z =   0.600 mm,
	W =180.000 deg,	P =   0.000 deg,	R =    90.000 deg
};
P[5823]{
   GP1:
	UF : 1, UT : 1,		CONFIG : 'N U T, 0, 0, 1',
	X =  115.000  mm,	Y =  109.000  mm,	Z =   15.000 mm,
	W =180.000 deg,	P =   0.000 deg,	R =    90.000 deg
};
P[5824]{
   GP1:
	UF : 1, UT : 1,		CONFIG : 'N U T, 0, 0, 1',
	X =  118.000  mm,	Y =  109.000  mm,	Z =   15.000 mm,
	W =180.000 deg,	P =   0.000 deg,	R =    90.000 deg
};
P[5825]{
   GP1:
	UF : 1, UT : 1,		CONFIG : 'N U T, 0, 0, 1',
	X =  118.000  mm,	Y =  109.000  mm,	Z =   0.600 mm,
	W =180.000 deg,	P =   0.000 deg,	R =    90.000 deg
};
P[5826]{
   GP1:
	UF : 1, UT : 1,		CONFIG : 'N U T, 0, 0, 1',
	X =  118.000  mm,	Y =  109.000  mm,	Z =   15.000 mm,
	W =180.000 deg,	P =   0.000 deg,	R =    90.000 deg
};
P[5842]{
   GP1:
	UF : 1, UT : 1,		CONFIG : 'N U T, 0, 0, 1',
	X =  136.000  mm,	Y =  109.000  mm,	Z =   15.000 mm,
	W =180.000 deg,	P =   0.000 deg,	R =    90.000 deg
};
P[5843]{
   GP1:
	UF : 1, UT : 1,		CONFIG : 'N U T, 0, 0, 1',
	X =  136.000  mm,	Y =  109.000  mm,	Z =   0.600 mm,
	W =180.000 deg,	P =   0.000 deg,	R =    90.000 deg
};
P[5844]{
   GP1:
	UF : 1, UT : 1,		CONFIG : 'N U T, 0, 0, 1',
	X =  136.000  mm,	Y =  109.000  mm,	Z =   15.000 mm,
	W =180.000 deg,	P =   0.000 deg,	R =    90.000 deg
};
P[5848]{
   GP1:
	UF : 1, UT : 1,		CONFIG : 'N U T, 0, 0, 1',
	X =  142.000  mm,	Y =  109.000  mm,	Z =   15.000 mm,
	W =180.000 deg,	P =   0.000 deg,	R =    90.000 deg
};
P[5849]{
   GP1:
	UF : 1, UT : 1,		CONFIG : 'N U T, 0, 0, 1',
	X =  142.000  mm,	Y =  109.000  mm,	Z =   0.600 mm,
	W =180.000 deg,	P =   0.000 deg,	R =    90.000 deg
};
P[5850]{
   GP1:
	UF : 1, UT : 1,		CONFIG : 'N U T, 0, 0, 1',
	X =  142.000  mm,	Y =  109.000  mm,	Z =   15.000 mm,
	W =180.000 deg,	P =   0.000 deg,	R =    90.000 deg
};
P[5851]{
   GP1:
	UF : 1, UT : 1,		CONFIG : 'N U T, 0, 0, 1',
	X =  160.000  mm,	Y =  109.000  mm,	Z =   15.000 mm,
	W =180.000 deg,	P =   0.000 deg,	R =    90.000 deg
};
P[5852]{
   GP1:
	UF : 1, UT : 1,		CONFIG : 'N U T, 0, 0, 1',
	X =  160.000  mm,	Y =  109.000  mm,	Z =   0.600 mm,
	W =180.000 deg,	P =   0.000 deg,	R =    90.000 deg
};
P[5853]{
   GP1:
	UF : 1, UT : 1,		CONFIG : 'N U T, 0, 0, 1',
	X =  160.000  mm,	Y =  109.000  mm,	Z =   15.000 mm,
	W =180.000 deg,	P =   0.000 deg,	R =    90.000 deg
};
P[5854]{
   GP1:
	UF : 1, UT : 1,		CONFIG : 'N U T, 0, 0, 1',
	X =  163.000  mm,	Y =  109.000  mm,	Z =   15.000 mm,
	W =180.000 deg,	P =   0.000 deg,	R =    90.000 deg
};
P[5855]{
   GP1:
	UF : 1, UT : 1,		CONFIG : 'N U T, 0, 0, 1',
	X =  163.000  mm,	Y =  109.000  mm,	Z =   0.600 mm,
	W =180.000 deg,	P =   0.000 deg,	R =    90.000 deg
};
P[5856]{
   GP1:
	UF : 1, UT : 1,		CONFIG : 'N U T, 0, 0, 1',
	X =  163.000  mm,	Y =  109.000  mm,	Z =   15.000 mm,
	W =180.000 deg,	P =   0.000 deg,	R =    90.000 deg
};
P[5857]{
   GP1:
	UF : 1, UT : 1,		CONFIG : 'N U T, 0, 0, 1',
	X =  166.000  mm,	Y =  109.000  mm,	Z =   15.000 mm,
	W =180.000 deg,	P =   0.000 deg,	R =    90.000 deg
};
P[5858]{
   GP1:
	UF : 1, UT : 1,		CONFIG : 'N U T, 0, 0, 1',
	X =  166.000  mm,	Y =  109.000  mm,	Z =   0.600 mm,
	W =180.000 deg,	P =   0.000 deg,	R =    90.000 deg
};
P[5859]{
   GP1:
	UF : 1, UT : 1,		CONFIG : 'N U T, 0, 0, 1',
	X =  166.000  mm,	Y =  109.000  mm,	Z =   15.000 mm,
	W =180.000 deg,	P =   0.000 deg,	R =    90.000 deg
};
P[5860]{
   GP1:
	UF : 1, UT : 1,		CONFIG : 'N U T, 0, 0, 1',
	X =  169.000  mm,	Y =  109.000  mm,	Z =   15.000 mm,
	W =180.000 deg,	P =   0.000 deg,	R =    90.000 deg
};
P[5861]{
   GP1:
	UF : 1, UT : 1,		CONFIG : 'N U T, 0, 0, 1',
	X =  169.000  mm,	Y =  109.000  mm,	Z =   0.600 mm,
	W =180.000 deg,	P =   0.000 deg,	R =    90.000 deg
};
P[5862]{
   GP1:
	UF : 1, UT : 1,		CONFIG : 'N U T, 0, 0, 1',
	X =  169.000  mm,	Y =  109.000  mm,	Z =   15.000 mm,
	W =180.000 deg,	P =   0.000 deg,	R =    90.000 deg
};
P[5863]{
   GP1:
	UF : 1, UT : 1,		CONFIG : 'N U T, 0, 0, 1',
	X =  172.000  mm,	Y =  109.000  mm,	Z =   15.000 mm,
	W =180.000 deg,	P =   0.000 deg,	R =    90.000 deg
};
P[5864]{
   GP1:
	UF : 1, UT : 1,		CONFIG : 'N U T, 0, 0, 1',
	X =  172.000  mm,	Y =  109.000  mm,	Z =   0.600 mm,
	W =180.000 deg,	P =   0.000 deg,	R =    90.000 deg
};
P[5865]{
   GP1:
	UF : 1, UT : 1,		CONFIG : 'N U T, 0, 0, 1',
	X =  172.000  mm,	Y =  109.000  mm,	Z =   15.000 mm,
	W =180.000 deg,	P =   0.000 deg,	R =    90.000 deg
};
P[5866]{
   GP1:
	UF : 1, UT : 1,		CONFIG : 'N U T, 0, 0, 1',
	X =  175.000  mm,	Y =  109.000  mm,	Z =   15.000 mm,
	W =180.000 deg,	P =   0.000 deg,	R =    90.000 deg
};
P[5867]{
   GP1:
	UF : 1, UT : 1,		CONFIG : 'N U T, 0, 0, 1',
	X =  175.000  mm,	Y =  109.000  mm,	Z =   0.600 mm,
	W =180.000 deg,	P =   0.000 deg,	R =    90.000 deg
};
P[5868]{
   GP1:
	UF : 1, UT : 1,		CONFIG : 'N U T, 0, 0, 1',
	X =  175.000  mm,	Y =  109.000  mm,	Z =   15.000 mm,
	W =180.000 deg,	P =   0.000 deg,	R =    90.000 deg
};
P[5869]{
   GP1:
	UF : 1, UT : 1,		CONFIG : 'N U T, 0, 0, 1',
	X =  178.000  mm,	Y =  109.000  mm,	Z =   15.000 mm,
	W =180.000 deg,	P =   0.000 deg,	R =    90.000 deg
};
P[5870]{
   GP1:
	UF : 1, UT : 1,		CONFIG : 'N U T, 0, 0, 1',
	X =  178.000  mm,	Y =  109.000  mm,	Z =   0.600 mm,
	W =180.000 deg,	P =   0.000 deg,	R =    90.000 deg
};
P[5871]{
   GP1:
	UF : 1, UT : 1,		CONFIG : 'N U T, 0, 0, 1',
	X =  178.000  mm,	Y =  109.000  mm,	Z =   15.000 mm,
	W =180.000 deg,	P =   0.000 deg,	R =    90.000 deg
};
P[5875]{
   GP1:
	UF : 1, UT : 1,		CONFIG : 'N U T, 0, 0, 1',
	X =  13.000  mm,	Y =  112.000  mm,	Z =   15.000 mm,
	W =180.000 deg,	P =   0.000 deg,	R =    90.000 deg
};
P[5876]{
   GP1:
	UF : 1, UT : 1,		CONFIG : 'N U T, 0, 0, 1',
	X =  13.000  mm,	Y =  112.000  mm,	Z =   0.600 mm,
	W =180.000 deg,	P =   0.000 deg,	R =    90.000 deg
};
P[5877]{
   GP1:
	UF : 1, UT : 1,		CONFIG : 'N U T, 0, 0, 1',
	X =  13.000  mm,	Y =  112.000  mm,	Z =   15.000 mm,
	W =180.000 deg,	P =   0.000 deg,	R =    90.000 deg
};
P[5878]{
   GP1:
	UF : 1, UT : 1,		CONFIG : 'N U T, 0, 0, 1',
	X =  16.000  mm,	Y =  112.000  mm,	Z =   15.000 mm,
	W =180.000 deg,	P =   0.000 deg,	R =    90.000 deg
};
P[5879]{
   GP1:
	UF : 1, UT : 1,		CONFIG : 'N U T, 0, 0, 1',
	X =  16.000  mm,	Y =  112.000  mm,	Z =   0.600 mm,
	W =180.000 deg,	P =   0.000 deg,	R =    90.000 deg
};
P[5880]{
   GP1:
	UF : 1, UT : 1,		CONFIG : 'N U T, 0, 0, 1',
	X =  16.000  mm,	Y =  112.000  mm,	Z =   15.000 mm,
	W =180.000 deg,	P =   0.000 deg,	R =    90.000 deg
};
P[5905]{
   GP1:
	UF : 1, UT : 1,		CONFIG : 'N U T, 0, 0, 1',
	X =  43.000  mm,	Y =  112.000  mm,	Z =   15.000 mm,
	W =180.000 deg,	P =   0.000 deg,	R =    90.000 deg
};
P[5906]{
   GP1:
	UF : 1, UT : 1,		CONFIG : 'N U T, 0, 0, 1',
	X =  43.000  mm,	Y =  112.000  mm,	Z =   0.600 mm,
	W =180.000 deg,	P =   0.000 deg,	R =    90.000 deg
};
P[5907]{
   GP1:
	UF : 1, UT : 1,		CONFIG : 'N U T, 0, 0, 1',
	X =  43.000  mm,	Y =  112.000  mm,	Z =   15.000 mm,
	W =180.000 deg,	P =   0.000 deg,	R =    90.000 deg
};
P[5920]{
   GP1:
	UF : 1, UT : 1,		CONFIG : 'N U T, 0, 0, 1',
	X =  115.000  mm,	Y =  112.000  mm,	Z =   15.000 mm,
	W =180.000 deg,	P =   0.000 deg,	R =    90.000 deg
};
P[5921]{
   GP1:
	UF : 1, UT : 1,		CONFIG : 'N U T, 0, 0, 1',
	X =  115.000  mm,	Y =  112.000  mm,	Z =   0.600 mm,
	W =180.000 deg,	P =   0.000 deg,	R =    90.000 deg
};
P[5922]{
   GP1:
	UF : 1, UT : 1,		CONFIG : 'N U T, 0, 0, 1',
	X =  115.000  mm,	Y =  112.000  mm,	Z =   15.000 mm,
	W =180.000 deg,	P =   0.000 deg,	R =    90.000 deg
};
P[5923]{
   GP1:
	UF : 1, UT : 1,		CONFIG : 'N U T, 0, 0, 1',
	X =  118.000  mm,	Y =  112.000  mm,	Z =   15.000 mm,
	W =180.000 deg,	P =   0.000 deg,	R =    90.000 deg
};
P[5924]{
   GP1:
	UF : 1, UT : 1,		CONFIG : 'N U T, 0, 0, 1',
	X =  118.000  mm,	Y =  112.000  mm,	Z =   0.600 mm,
	W =180.000 deg,	P =   0.000 deg,	R =    90.000 deg
};
P[5925]{
   GP1:
	UF : 1, UT : 1,		CONFIG : 'N U T, 0, 0, 1',
	X =  118.000  mm,	Y =  112.000  mm,	Z =   15.000 mm,
	W =180.000 deg,	P =   0.000 deg,	R =    90.000 deg
};
P[5932]{
   GP1:
	UF : 1, UT : 1,		CONFIG : 'N U T, 0, 0, 1',
	X =  127.000  mm,	Y =  112.000  mm,	Z =   15.000 mm,
	W =180.000 deg,	P =   0.000 deg,	R =    90.000 deg
};
P[5933]{
   GP1:
	UF : 1, UT : 1,		CONFIG : 'N U T, 0, 0, 1',
	X =  127.000  mm,	Y =  112.000  mm,	Z =   0.600 mm,
	W =180.000 deg,	P =   0.000 deg,	R =    90.000 deg
};
P[5934]{
   GP1:
	UF : 1, UT : 1,		CONFIG : 'N U T, 0, 0, 1',
	X =  127.000  mm,	Y =  112.000  mm,	Z =   15.000 mm,
	W =180.000 deg,	P =   0.000 deg,	R =    90.000 deg
};
P[5935]{
   GP1:
	UF : 1, UT : 1,		CONFIG : 'N U T, 0, 0, 1',
	X =  130.000  mm,	Y =  112.000  mm,	Z =   15.000 mm,
	W =180.000 deg,	P =   0.000 deg,	R =    90.000 deg
};
P[5936]{
   GP1:
	UF : 1, UT : 1,		CONFIG : 'N U T, 0, 0, 1',
	X =  130.000  mm,	Y =  112.000  mm,	Z =   0.600 mm,
	W =180.000 deg,	P =   0.000 deg,	R =    90.000 deg
};
P[5937]{
   GP1:
	UF : 1, UT : 1,		CONFIG : 'N U T, 0, 0, 1',
	X =  130.000  mm,	Y =  112.000  mm,	Z =   15.000 mm,
	W =180.000 deg,	P =   0.000 deg,	R =    90.000 deg
};
P[5938]{
   GP1:
	UF : 1, UT : 1,		CONFIG : 'N U T, 0, 0, 1',
	X =  133.000  mm,	Y =  112.000  mm,	Z =   15.000 mm,
	W =180.000 deg,	P =   0.000 deg,	R =    90.000 deg
};
P[5939]{
   GP1:
	UF : 1, UT : 1,		CONFIG : 'N U T, 0, 0, 1',
	X =  133.000  mm,	Y =  112.000  mm,	Z =   0.600 mm,
	W =180.000 deg,	P =   0.000 deg,	R =    90.000 deg
};
P[5940]{
   GP1:
	UF : 1, UT : 1,		CONFIG : 'N U T, 0, 0, 1',
	X =  133.000  mm,	Y =  112.000  mm,	Z =   15.000 mm,
	W =180.000 deg,	P =   0.000 deg,	R =    90.000 deg
};
P[5941]{
   GP1:
	UF : 1, UT : 1,		CONFIG : 'N U T, 0, 0, 1',
	X =  136.000  mm,	Y =  112.000  mm,	Z =   15.000 mm,
	W =180.000 deg,	P =   0.000 deg,	R =    90.000 deg
};
P[5942]{
   GP1:
	UF : 1, UT : 1,		CONFIG : 'N U T, 0, 0, 1',
	X =  136.000  mm,	Y =  112.000  mm,	Z =   0.600 mm,
	W =180.000 deg,	P =   0.000 deg,	R =    90.000 deg
};
P[5943]{
   GP1:
	UF : 1, UT : 1,		CONFIG : 'N U T, 0, 0, 1',
	X =  136.000  mm,	Y =  112.000  mm,	Z =   15.000 mm,
	W =180.000 deg,	P =   0.000 deg,	R =    90.000 deg
};
P[5944]{
   GP1:
	UF : 1, UT : 1,		CONFIG : 'N U T, 0, 0, 1',
	X =  139.000  mm,	Y =  112.000  mm,	Z =   15.000 mm,
	W =180.000 deg,	P =   0.000 deg,	R =    90.000 deg
};
P[5945]{
   GP1:
	UF : 1, UT : 1,		CONFIG : 'N U T, 0, 0, 1',
	X =  139.000  mm,	Y =  112.000  mm,	Z =   0.600 mm,
	W =180.000 deg,	P =   0.000 deg,	R =    90.000 deg
};
P[5946]{
   GP1:
	UF : 1, UT : 1,		CONFIG : 'N U T, 0, 0, 1',
	X =  139.000  mm,	Y =  112.000  mm,	Z =   15.000 mm,
	W =180.000 deg,	P =   0.000 deg,	R =    90.000 deg
};
P[5947]{
   GP1:
	UF : 1, UT : 1,		CONFIG : 'N U T, 0, 0, 1',
	X =  160.000  mm,	Y =  112.000  mm,	Z =   15.000 mm,
	W =180.000 deg,	P =   0.000 deg,	R =    90.000 deg
};
P[5948]{
   GP1:
	UF : 1, UT : 1,		CONFIG : 'N U T, 0, 0, 1',
	X =  160.000  mm,	Y =  112.000  mm,	Z =   0.600 mm,
	W =180.000 deg,	P =   0.000 deg,	R =    90.000 deg
};
P[5949]{
   GP1:
	UF : 1, UT : 1,		CONFIG : 'N U T, 0, 0, 1',
	X =  160.000  mm,	Y =  112.000  mm,	Z =   15.000 mm,
	W =180.000 deg,	P =   0.000 deg,	R =    90.000 deg
};
P[5950]{
   GP1:
	UF : 1, UT : 1,		CONFIG : 'N U T, 0, 0, 1',
	X =  163.000  mm,	Y =  112.000  mm,	Z =   15.000 mm,
	W =180.000 deg,	P =   0.000 deg,	R =    90.000 deg
};
P[5951]{
   GP1:
	UF : 1, UT : 1,		CONFIG : 'N U T, 0, 0, 1',
	X =  163.000  mm,	Y =  112.000  mm,	Z =   0.600 mm,
	W =180.000 deg,	P =   0.000 deg,	R =    90.000 deg
};
P[5952]{
   GP1:
	UF : 1, UT : 1,		CONFIG : 'N U T, 0, 0, 1',
	X =  163.000  mm,	Y =  112.000  mm,	Z =   15.000 mm,
	W =180.000 deg,	P =   0.000 deg,	R =    90.000 deg
};
P[5953]{
   GP1:
	UF : 1, UT : 1,		CONFIG : 'N U T, 0, 0, 1',
	X =  166.000  mm,	Y =  112.000  mm,	Z =   15.000 mm,
	W =180.000 deg,	P =   0.000 deg,	R =    90.000 deg
};
P[5954]{
   GP1:
	UF : 1, UT : 1,		CONFIG : 'N U T, 0, 0, 1',
	X =  166.000  mm,	Y =  112.000  mm,	Z =   0.600 mm,
	W =180.000 deg,	P =   0.000 deg,	R =    90.000 deg
};
P[5955]{
   GP1:
	UF : 1, UT : 1,		CONFIG : 'N U T, 0, 0, 1',
	X =  166.000  mm,	Y =  112.000  mm,	Z =   15.000 mm,
	W =180.000 deg,	P =   0.000 deg,	R =    90.000 deg
};
P[5956]{
   GP1:
	UF : 1, UT : 1,		CONFIG : 'N U T, 0, 0, 1',
	X =  169.000  mm,	Y =  112.000  mm,	Z =   15.000 mm,
	W =180.000 deg,	P =   0.000 deg,	R =    90.000 deg
};
P[5957]{
   GP1:
	UF : 1, UT : 1,		CONFIG : 'N U T, 0, 0, 1',
	X =  169.000  mm,	Y =  112.000  mm,	Z =   0.600 mm,
	W =180.000 deg,	P =   0.000 deg,	R =    90.000 deg
};
P[5958]{
   GP1:
	UF : 1, UT : 1,		CONFIG : 'N U T, 0, 0, 1',
	X =  169.000  mm,	Y =  112.000  mm,	Z =   15.000 mm,
	W =180.000 deg,	P =   0.000 deg,	R =    90.000 deg
};
P[5959]{
   GP1:
	UF : 1, UT : 1,		CONFIG : 'N U T, 0, 0, 1',
	X =  172.000  mm,	Y =  112.000  mm,	Z =   15.000 mm,
	W =180.000 deg,	P =   0.000 deg,	R =    90.000 deg
};
P[5960]{
   GP1:
	UF : 1, UT : 1,		CONFIG : 'N U T, 0, 0, 1',
	X =  172.000  mm,	Y =  112.000  mm,	Z =   0.600 mm,
	W =180.000 deg,	P =   0.000 deg,	R =    90.000 deg
};
P[5961]{
   GP1:
	UF : 1, UT : 1,		CONFIG : 'N U T, 0, 0, 1',
	X =  172.000  mm,	Y =  112.000  mm,	Z =   15.000 mm,
	W =180.000 deg,	P =   0.000 deg,	R =    90.000 deg
};
P[5962]{
   GP1:
	UF : 1, UT : 1,		CONFIG : 'N U T, 0, 0, 1',
	X =  175.000  mm,	Y =  112.000  mm,	Z =   15.000 mm,
	W =180.000 deg,	P =   0.000 deg,	R =    90.000 deg
};
P[5963]{
   GP1:
	UF : 1, UT : 1,		CONFIG : 'N U T, 0, 0, 1',
	X =  175.000  mm,	Y =  112.000  mm,	Z =   0.600 mm,
	W =180.000 deg,	P =   0.000 deg,	R =    90.000 deg
};
P[5964]{
   GP1:
	UF : 1, UT : 1,		CONFIG : 'N U T, 0, 0, 1',
	X =  175.000  mm,	Y =  112.000  mm,	Z =   15.000 mm,
	W =180.000 deg,	P =   0.000 deg,	R =    90.000 deg
};
P[5965]{
   GP1:
	UF : 1, UT : 1,		CONFIG : 'N U T, 0, 0, 1',
	X =  178.000  mm,	Y =  112.000  mm,	Z =   15.000 mm,
	W =180.000 deg,	P =   0.000 deg,	R =    90.000 deg
};
P[5966]{
   GP1:
	UF : 1, UT : 1,		CONFIG : 'N U T, 0, 0, 1',
	X =  178.000  mm,	Y =  112.000  mm,	Z =   0.600 mm,
	W =180.000 deg,	P =   0.000 deg,	R =    90.000 deg
};
P[5967]{
   GP1:
	UF : 1, UT : 1,		CONFIG : 'N U T, 0, 0, 1',
	X =  178.000  mm,	Y =  112.000  mm,	Z =   15.000 mm,
	W =180.000 deg,	P =   0.000 deg,	R =    90.000 deg
};
P[5974]{
   GP1:
	UF : 1, UT : 1,		CONFIG : 'N U T, 0, 0, 1',
	X =  25.000  mm,	Y =  115.000  mm,	Z =   15.000 mm,
	W =180.000 deg,	P =   0.000 deg,	R =    90.000 deg
};
P[5975]{
   GP1:
	UF : 1, UT : 1,		CONFIG : 'N U T, 0, 0, 1',
	X =  25.000  mm,	Y =  115.000  mm,	Z =   0.600 mm,
	W =180.000 deg,	P =   0.000 deg,	R =    90.000 deg
};
P[5976]{
   GP1:
	UF : 1, UT : 1,		CONFIG : 'N U T, 0, 0, 1',
	X =  25.000  mm,	Y =  115.000  mm,	Z =   15.000 mm,
	W =180.000 deg,	P =   0.000 deg,	R =    90.000 deg
};
P[5977]{
   GP1:
	UF : 1, UT : 1,		CONFIG : 'N U T, 0, 0, 1',
	X =  28.000  mm,	Y =  115.000  mm,	Z =   15.000 mm,
	W =180.000 deg,	P =   0.000 deg,	R =    90.000 deg
};
P[5978]{
   GP1:
	UF : 1, UT : 1,		CONFIG : 'N U T, 0, 0, 1',
	X =  28.000  mm,	Y =  115.000  mm,	Z =   0.600 mm,
	W =180.000 deg,	P =   0.000 deg,	R =    90.000 deg
};
P[5979]{
   GP1:
	UF : 1, UT : 1,		CONFIG : 'N U T, 0, 0, 1',
	X =  28.000  mm,	Y =  115.000  mm,	Z =   15.000 mm,
	W =180.000 deg,	P =   0.000 deg,	R =    90.000 deg
};
P[5980]{
   GP1:
	UF : 1, UT : 1,		CONFIG : 'N U T, 0, 0, 1',
	X =  31.000  mm,	Y =  115.000  mm,	Z =   15.000 mm,
	W =180.000 deg,	P =   0.000 deg,	R =    90.000 deg
};
P[5981]{
   GP1:
	UF : 1, UT : 1,		CONFIG : 'N U T, 0, 0, 1',
	X =  31.000  mm,	Y =  115.000  mm,	Z =   0.600 mm,
	W =180.000 deg,	P =   0.000 deg,	R =    90.000 deg
};
P[5982]{
   GP1:
	UF : 1, UT : 1,		CONFIG : 'N U T, 0, 0, 1',
	X =  31.000  mm,	Y =  115.000  mm,	Z =   15.000 mm,
	W =180.000 deg,	P =   0.000 deg,	R =    90.000 deg
};
P[5983]{
   GP1:
	UF : 1, UT : 1,		CONFIG : 'N U T, 0, 0, 1',
	X =  34.000  mm,	Y =  115.000  mm,	Z =   15.000 mm,
	W =180.000 deg,	P =   0.000 deg,	R =    90.000 deg
};
P[5984]{
   GP1:
	UF : 1, UT : 1,		CONFIG : 'N U T, 0, 0, 1',
	X =  34.000  mm,	Y =  115.000  mm,	Z =   0.600 mm,
	W =180.000 deg,	P =   0.000 deg,	R =    90.000 deg
};
P[5985]{
   GP1:
	UF : 1, UT : 1,		CONFIG : 'N U T, 0, 0, 1',
	X =  34.000  mm,	Y =  115.000  mm,	Z =   15.000 mm,
	W =180.000 deg,	P =   0.000 deg,	R =    90.000 deg
};
P[5986]{
   GP1:
	UF : 1, UT : 1,		CONFIG : 'N U T, 0, 0, 1',
	X =  37.000  mm,	Y =  115.000  mm,	Z =   15.000 mm,
	W =180.000 deg,	P =   0.000 deg,	R =    90.000 deg
};
P[5987]{
   GP1:
	UF : 1, UT : 1,		CONFIG : 'N U T, 0, 0, 1',
	X =  37.000  mm,	Y =  115.000  mm,	Z =   0.600 mm,
	W =180.000 deg,	P =   0.000 deg,	R =    90.000 deg
};
P[5988]{
   GP1:
	UF : 1, UT : 1,		CONFIG : 'N U T, 0, 0, 1',
	X =  37.000  mm,	Y =  115.000  mm,	Z =   15.000 mm,
	W =180.000 deg,	P =   0.000 deg,	R =    90.000 deg
};
P[6013]{
   GP1:
	UF : 1, UT : 1,		CONFIG : 'N U T, 0, 0, 1',
	X =  121.000  mm,	Y =  115.000  mm,	Z =   15.000 mm,
	W =180.000 deg,	P =   0.000 deg,	R =    90.000 deg
};
P[6014]{
   GP1:
	UF : 1, UT : 1,		CONFIG : 'N U T, 0, 0, 1',
	X =  121.000  mm,	Y =  115.000  mm,	Z =   0.600 mm,
	W =180.000 deg,	P =   0.000 deg,	R =    90.000 deg
};
P[6015]{
   GP1:
	UF : 1, UT : 1,		CONFIG : 'N U T, 0, 0, 1',
	X =  121.000  mm,	Y =  115.000  mm,	Z =   15.000 mm,
	W =180.000 deg,	P =   0.000 deg,	R =    90.000 deg
};
P[6016]{
   GP1:
	UF : 1, UT : 1,		CONFIG : 'N U T, 0, 0, 1',
	X =  124.000  mm,	Y =  115.000  mm,	Z =   15.000 mm,
	W =180.000 deg,	P =   0.000 deg,	R =    90.000 deg
};
P[6017]{
   GP1:
	UF : 1, UT : 1,		CONFIG : 'N U T, 0, 0, 1',
	X =  124.000  mm,	Y =  115.000  mm,	Z =   0.600 mm,
	W =180.000 deg,	P =   0.000 deg,	R =    90.000 deg
};
P[6018]{
   GP1:
	UF : 1, UT : 1,		CONFIG : 'N U T, 0, 0, 1',
	X =  124.000  mm,	Y =  115.000  mm,	Z =   15.000 mm,
	W =180.000 deg,	P =   0.000 deg,	R =    90.000 deg
};
P[6019]{
   GP1:
	UF : 1, UT : 1,		CONFIG : 'N U T, 0, 0, 1',
	X =  127.000  mm,	Y =  115.000  mm,	Z =   15.000 mm,
	W =180.000 deg,	P =   0.000 deg,	R =    90.000 deg
};
P[6020]{
   GP1:
	UF : 1, UT : 1,		CONFIG : 'N U T, 0, 0, 1',
	X =  127.000  mm,	Y =  115.000  mm,	Z =   0.600 mm,
	W =180.000 deg,	P =   0.000 deg,	R =    90.000 deg
};
P[6021]{
   GP1:
	UF : 1, UT : 1,		CONFIG : 'N U T, 0, 0, 1',
	X =  127.000  mm,	Y =  115.000  mm,	Z =   15.000 mm,
	W =180.000 deg,	P =   0.000 deg,	R =    90.000 deg
};
P[6022]{
   GP1:
	UF : 1, UT : 1,		CONFIG : 'N U T, 0, 0, 1',
	X =  130.000  mm,	Y =  115.000  mm,	Z =   15.000 mm,
	W =180.000 deg,	P =   0.000 deg,	R =    90.000 deg
};
P[6023]{
   GP1:
	UF : 1, UT : 1,		CONFIG : 'N U T, 0, 0, 1',
	X =  130.000  mm,	Y =  115.000  mm,	Z =   0.600 mm,
	W =180.000 deg,	P =   0.000 deg,	R =    90.000 deg
};
P[6024]{
   GP1:
	UF : 1, UT : 1,		CONFIG : 'N U T, 0, 0, 1',
	X =  130.000  mm,	Y =  115.000  mm,	Z =   15.000 mm,
	W =180.000 deg,	P =   0.000 deg,	R =    90.000 deg
};
P[6025]{
   GP1:
	UF : 1, UT : 1,		CONFIG : 'N U T, 0, 0, 1',
	X =  133.000  mm,	Y =  115.000  mm,	Z =   15.000 mm,
	W =180.000 deg,	P =   0.000 deg,	R =    90.000 deg
};
P[6026]{
   GP1:
	UF : 1, UT : 1,		CONFIG : 'N U T, 0, 0, 1',
	X =  133.000  mm,	Y =  115.000  mm,	Z =   0.600 mm,
	W =180.000 deg,	P =   0.000 deg,	R =    90.000 deg
};
P[6027]{
   GP1:
	UF : 1, UT : 1,		CONFIG : 'N U T, 0, 0, 1',
	X =  133.000  mm,	Y =  115.000  mm,	Z =   15.000 mm,
	W =180.000 deg,	P =   0.000 deg,	R =    90.000 deg
};
P[6028]{
   GP1:
	UF : 1, UT : 1,		CONFIG : 'N U T, 0, 0, 1',
	X =  136.000  mm,	Y =  115.000  mm,	Z =   15.000 mm,
	W =180.000 deg,	P =   0.000 deg,	R =    90.000 deg
};
P[6029]{
   GP1:
	UF : 1, UT : 1,		CONFIG : 'N U T, 0, 0, 1',
	X =  136.000  mm,	Y =  115.000  mm,	Z =   0.600 mm,
	W =180.000 deg,	P =   0.000 deg,	R =    90.000 deg
};
P[6030]{
   GP1:
	UF : 1, UT : 1,		CONFIG : 'N U T, 0, 0, 1',
	X =  136.000  mm,	Y =  115.000  mm,	Z =   15.000 mm,
	W =180.000 deg,	P =   0.000 deg,	R =    90.000 deg
};
P[6031]{
   GP1:
	UF : 1, UT : 1,		CONFIG : 'N U T, 0, 0, 1',
	X =  139.000  mm,	Y =  115.000  mm,	Z =   15.000 mm,
	W =180.000 deg,	P =   0.000 deg,	R =    90.000 deg
};
P[6032]{
   GP1:
	UF : 1, UT : 1,		CONFIG : 'N U T, 0, 0, 1',
	X =  139.000  mm,	Y =  115.000  mm,	Z =   0.600 mm,
	W =180.000 deg,	P =   0.000 deg,	R =    90.000 deg
};
P[6033]{
   GP1:
	UF : 1, UT : 1,		CONFIG : 'N U T, 0, 0, 1',
	X =  139.000  mm,	Y =  115.000  mm,	Z =   15.000 mm,
	W =180.000 deg,	P =   0.000 deg,	R =    90.000 deg
};
P[6037]{
   GP1:
	UF : 1, UT : 1,		CONFIG : 'N U T, 0, 0, 1',
	X =  160.000  mm,	Y =  115.000  mm,	Z =   15.000 mm,
	W =180.000 deg,	P =   0.000 deg,	R =    90.000 deg
};
P[6038]{
   GP1:
	UF : 1, UT : 1,		CONFIG : 'N U T, 0, 0, 1',
	X =  160.000  mm,	Y =  115.000  mm,	Z =   0.600 mm,
	W =180.000 deg,	P =   0.000 deg,	R =    90.000 deg
};
P[6039]{
   GP1:
	UF : 1, UT : 1,		CONFIG : 'N U T, 0, 0, 1',
	X =  160.000  mm,	Y =  115.000  mm,	Z =   15.000 mm,
	W =180.000 deg,	P =   0.000 deg,	R =    90.000 deg
};
P[6040]{
   GP1:
	UF : 1, UT : 1,		CONFIG : 'N U T, 0, 0, 1',
	X =  163.000  mm,	Y =  115.000  mm,	Z =   15.000 mm,
	W =180.000 deg,	P =   0.000 deg,	R =    90.000 deg
};
P[6041]{
   GP1:
	UF : 1, UT : 1,		CONFIG : 'N U T, 0, 0, 1',
	X =  163.000  mm,	Y =  115.000  mm,	Z =   0.600 mm,
	W =180.000 deg,	P =   0.000 deg,	R =    90.000 deg
};
P[6042]{
   GP1:
	UF : 1, UT : 1,		CONFIG : 'N U T, 0, 0, 1',
	X =  163.000  mm,	Y =  115.000  mm,	Z =   15.000 mm,
	W =180.000 deg,	P =   0.000 deg,	R =    90.000 deg
};
P[6043]{
   GP1:
	UF : 1, UT : 1,		CONFIG : 'N U T, 0, 0, 1',
	X =  166.000  mm,	Y =  115.000  mm,	Z =   15.000 mm,
	W =180.000 deg,	P =   0.000 deg,	R =    90.000 deg
};
P[6044]{
   GP1:
	UF : 1, UT : 1,		CONFIG : 'N U T, 0, 0, 1',
	X =  166.000  mm,	Y =  115.000  mm,	Z =   0.600 mm,
	W =180.000 deg,	P =   0.000 deg,	R =    90.000 deg
};
P[6045]{
   GP1:
	UF : 1, UT : 1,		CONFIG : 'N U T, 0, 0, 1',
	X =  166.000  mm,	Y =  115.000  mm,	Z =   15.000 mm,
	W =180.000 deg,	P =   0.000 deg,	R =    90.000 deg
};
P[6046]{
   GP1:
	UF : 1, UT : 1,		CONFIG : 'N U T, 0, 0, 1',
	X =  169.000  mm,	Y =  115.000  mm,	Z =   15.000 mm,
	W =180.000 deg,	P =   0.000 deg,	R =    90.000 deg
};
P[6047]{
   GP1:
	UF : 1, UT : 1,		CONFIG : 'N U T, 0, 0, 1',
	X =  169.000  mm,	Y =  115.000  mm,	Z =   0.600 mm,
	W =180.000 deg,	P =   0.000 deg,	R =    90.000 deg
};
P[6048]{
   GP1:
	UF : 1, UT : 1,		CONFIG : 'N U T, 0, 0, 1',
	X =  169.000  mm,	Y =  115.000  mm,	Z =   15.000 mm,
	W =180.000 deg,	P =   0.000 deg,	R =    90.000 deg
};
P[6049]{
   GP1:
	UF : 1, UT : 1,		CONFIG : 'N U T, 0, 0, 1',
	X =  172.000  mm,	Y =  115.000  mm,	Z =   15.000 mm,
	W =180.000 deg,	P =   0.000 deg,	R =    90.000 deg
};
P[6050]{
   GP1:
	UF : 1, UT : 1,		CONFIG : 'N U T, 0, 0, 1',
	X =  172.000  mm,	Y =  115.000  mm,	Z =   0.600 mm,
	W =180.000 deg,	P =   0.000 deg,	R =    90.000 deg
};
P[6051]{
   GP1:
	UF : 1, UT : 1,		CONFIG : 'N U T, 0, 0, 1',
	X =  172.000  mm,	Y =  115.000  mm,	Z =   15.000 mm,
	W =180.000 deg,	P =   0.000 deg,	R =    90.000 deg
};
P[6052]{
   GP1:
	UF : 1, UT : 1,		CONFIG : 'N U T, 0, 0, 1',
	X =  175.000  mm,	Y =  115.000  mm,	Z =   15.000 mm,
	W =180.000 deg,	P =   0.000 deg,	R =    90.000 deg
};
P[6053]{
   GP1:
	UF : 1, UT : 1,		CONFIG : 'N U T, 0, 0, 1',
	X =  175.000  mm,	Y =  115.000  mm,	Z =   0.600 mm,
	W =180.000 deg,	P =   0.000 deg,	R =    90.000 deg
};
P[6054]{
   GP1:
	UF : 1, UT : 1,		CONFIG : 'N U T, 0, 0, 1',
	X =  175.000  mm,	Y =  115.000  mm,	Z =   15.000 mm,
	W =180.000 deg,	P =   0.000 deg,	R =    90.000 deg
};
P[6055]{
   GP1:
	UF : 1, UT : 1,		CONFIG : 'N U T, 0, 0, 1',
	X =  178.000  mm,	Y =  115.000  mm,	Z =   15.000 mm,
	W =180.000 deg,	P =   0.000 deg,	R =    90.000 deg
};
P[6056]{
   GP1:
	UF : 1, UT : 1,		CONFIG : 'N U T, 0, 0, 1',
	X =  178.000  mm,	Y =  115.000  mm,	Z =   0.600 mm,
	W =180.000 deg,	P =   0.000 deg,	R =    90.000 deg
};
P[6057]{
   GP1:
	UF : 1, UT : 1,		CONFIG : 'N U T, 0, 0, 1',
	X =  178.000  mm,	Y =  115.000  mm,	Z =   15.000 mm,
	W =180.000 deg,	P =   0.000 deg,	R =    90.000 deg
};
P[6067]{
   GP1:
	UF : 1, UT : 1,		CONFIG : 'N U T, 0, 0, 1',
	X =  25.000  mm,	Y =  118.000  mm,	Z =   15.000 mm,
	W =180.000 deg,	P =   0.000 deg,	R =    90.000 deg
};
P[6068]{
   GP1:
	UF : 1, UT : 1,		CONFIG : 'N U T, 0, 0, 1',
	X =  25.000  mm,	Y =  118.000  mm,	Z =   0.600 mm,
	W =180.000 deg,	P =   0.000 deg,	R =    90.000 deg
};
P[6069]{
   GP1:
	UF : 1, UT : 1,		CONFIG : 'N U T, 0, 0, 1',
	X =  25.000  mm,	Y =  118.000  mm,	Z =   15.000 mm,
	W =180.000 deg,	P =   0.000 deg,	R =    90.000 deg
};
P[6106]{
   GP1:
	UF : 1, UT : 1,		CONFIG : 'N U T, 0, 0, 1',
	X =  118.000  mm,	Y =  118.000  mm,	Z =   15.000 mm,
	W =180.000 deg,	P =   0.000 deg,	R =    90.000 deg
};
P[6107]{
   GP1:
	UF : 1, UT : 1,		CONFIG : 'N U T, 0, 0, 1',
	X =  118.000  mm,	Y =  118.000  mm,	Z =   0.600 mm,
	W =180.000 deg,	P =   0.000 deg,	R =    90.000 deg
};
P[6108]{
   GP1:
	UF : 1, UT : 1,		CONFIG : 'N U T, 0, 0, 1',
	X =  118.000  mm,	Y =  118.000  mm,	Z =   15.000 mm,
	W =180.000 deg,	P =   0.000 deg,	R =    90.000 deg
};
P[6109]{
   GP1:
	UF : 1, UT : 1,		CONFIG : 'N U T, 0, 0, 1',
	X =  121.000  mm,	Y =  118.000  mm,	Z =   15.000 mm,
	W =180.000 deg,	P =   0.000 deg,	R =    90.000 deg
};
P[6110]{
   GP1:
	UF : 1, UT : 1,		CONFIG : 'N U T, 0, 0, 1',
	X =  121.000  mm,	Y =  118.000  mm,	Z =   0.600 mm,
	W =180.000 deg,	P =   0.000 deg,	R =    90.000 deg
};
P[6111]{
   GP1:
	UF : 1, UT : 1,		CONFIG : 'N U T, 0, 0, 1',
	X =  121.000  mm,	Y =  118.000  mm,	Z =   15.000 mm,
	W =180.000 deg,	P =   0.000 deg,	R =    90.000 deg
};
P[6112]{
   GP1:
	UF : 1, UT : 1,		CONFIG : 'N U T, 0, 0, 1',
	X =  124.000  mm,	Y =  118.000  mm,	Z =   15.000 mm,
	W =180.000 deg,	P =   0.000 deg,	R =    90.000 deg
};
P[6113]{
   GP1:
	UF : 1, UT : 1,		CONFIG : 'N U T, 0, 0, 1',
	X =  124.000  mm,	Y =  118.000  mm,	Z =   0.600 mm,
	W =180.000 deg,	P =   0.000 deg,	R =    90.000 deg
};
P[6114]{
   GP1:
	UF : 1, UT : 1,		CONFIG : 'N U T, 0, 0, 1',
	X =  124.000  mm,	Y =  118.000  mm,	Z =   15.000 mm,
	W =180.000 deg,	P =   0.000 deg,	R =    90.000 deg
};
P[6115]{
   GP1:
	UF : 1, UT : 1,		CONFIG : 'N U T, 0, 0, 1',
	X =  127.000  mm,	Y =  118.000  mm,	Z =   15.000 mm,
	W =180.000 deg,	P =   0.000 deg,	R =    90.000 deg
};
P[6116]{
   GP1:
	UF : 1, UT : 1,		CONFIG : 'N U T, 0, 0, 1',
	X =  127.000  mm,	Y =  118.000  mm,	Z =   0.600 mm,
	W =180.000 deg,	P =   0.000 deg,	R =    90.000 deg
};
P[6117]{
   GP1:
	UF : 1, UT : 1,		CONFIG : 'N U T, 0, 0, 1',
	X =  127.000  mm,	Y =  118.000  mm,	Z =   15.000 mm,
	W =180.000 deg,	P =   0.000 deg,	R =    90.000 deg
};
P[6118]{
   GP1:
	UF : 1, UT : 1,		CONFIG : 'N U T, 0, 0, 1',
	X =  130.000  mm,	Y =  118.000  mm,	Z =   15.000 mm,
	W =180.000 deg,	P =   0.000 deg,	R =    90.000 deg
};
P[6119]{
   GP1:
	UF : 1, UT : 1,		CONFIG : 'N U T, 0, 0, 1',
	X =  130.000  mm,	Y =  118.000  mm,	Z =   0.600 mm,
	W =180.000 deg,	P =   0.000 deg,	R =    90.000 deg
};
P[6120]{
   GP1:
	UF : 1, UT : 1,		CONFIG : 'N U T, 0, 0, 1',
	X =  130.000  mm,	Y =  118.000  mm,	Z =   15.000 mm,
	W =180.000 deg,	P =   0.000 deg,	R =    90.000 deg
};
P[6121]{
   GP1:
	UF : 1, UT : 1,		CONFIG : 'N U T, 0, 0, 1',
	X =  133.000  mm,	Y =  118.000  mm,	Z =   15.000 mm,
	W =180.000 deg,	P =   0.000 deg,	R =    90.000 deg
};
P[6122]{
   GP1:
	UF : 1, UT : 1,		CONFIG : 'N U T, 0, 0, 1',
	X =  133.000  mm,	Y =  118.000  mm,	Z =   0.600 mm,
	W =180.000 deg,	P =   0.000 deg,	R =    90.000 deg
};
P[6123]{
   GP1:
	UF : 1, UT : 1,		CONFIG : 'N U T, 0, 0, 1',
	X =  133.000  mm,	Y =  118.000  mm,	Z =   15.000 mm,
	W =180.000 deg,	P =   0.000 deg,	R =    90.000 deg
};
P[6124]{
   GP1:
	UF : 1, UT : 1,		CONFIG : 'N U T, 0, 0, 1',
	X =  136.000  mm,	Y =  118.000  mm,	Z =   15.000 mm,
	W =180.000 deg,	P =   0.000 deg,	R =    90.000 deg
};
P[6125]{
   GP1:
	UF : 1, UT : 1,		CONFIG : 'N U T, 0, 0, 1',
	X =  136.000  mm,	Y =  118.000  mm,	Z =   0.600 mm,
	W =180.000 deg,	P =   0.000 deg,	R =    90.000 deg
};
P[6126]{
   GP1:
	UF : 1, UT : 1,		CONFIG : 'N U T, 0, 0, 1',
	X =  136.000  mm,	Y =  118.000  mm,	Z =   15.000 mm,
	W =180.000 deg,	P =   0.000 deg,	R =    90.000 deg
};
P[6127]{
   GP1:
	UF : 1, UT : 1,		CONFIG : 'N U T, 0, 0, 1',
	X =  139.000  mm,	Y =  118.000  mm,	Z =   15.000 mm,
	W =180.000 deg,	P =   0.000 deg,	R =    90.000 deg
};
P[6128]{
   GP1:
	UF : 1, UT : 1,		CONFIG : 'N U T, 0, 0, 1',
	X =  139.000  mm,	Y =  118.000  mm,	Z =   0.600 mm,
	W =180.000 deg,	P =   0.000 deg,	R =    90.000 deg
};
P[6129]{
   GP1:
	UF : 1, UT : 1,		CONFIG : 'N U T, 0, 0, 1',
	X =  139.000  mm,	Y =  118.000  mm,	Z =   15.000 mm,
	W =180.000 deg,	P =   0.000 deg,	R =    90.000 deg
};
P[6130]{
   GP1:
	UF : 1, UT : 1,		CONFIG : 'N U T, 0, 0, 1',
	X =  142.000  mm,	Y =  118.000  mm,	Z =   15.000 mm,
	W =180.000 deg,	P =   0.000 deg,	R =    90.000 deg
};
P[6131]{
   GP1:
	UF : 1, UT : 1,		CONFIG : 'N U T, 0, 0, 1',
	X =  142.000  mm,	Y =  118.000  mm,	Z =   0.600 mm,
	W =180.000 deg,	P =   0.000 deg,	R =    90.000 deg
};
P[6132]{
   GP1:
	UF : 1, UT : 1,		CONFIG : 'N U T, 0, 0, 1',
	X =  142.000  mm,	Y =  118.000  mm,	Z =   15.000 mm,
	W =180.000 deg,	P =   0.000 deg,	R =    90.000 deg
};
P[6136]{
   GP1:
	UF : 1, UT : 1,		CONFIG : 'N U T, 0, 0, 1',
	X =  157.000  mm,	Y =  118.000  mm,	Z =   15.000 mm,
	W =180.000 deg,	P =   0.000 deg,	R =    90.000 deg
};
P[6137]{
   GP1:
	UF : 1, UT : 1,		CONFIG : 'N U T, 0, 0, 1',
	X =  157.000  mm,	Y =  118.000  mm,	Z =   0.600 mm,
	W =180.000 deg,	P =   0.000 deg,	R =    90.000 deg
};
P[6138]{
   GP1:
	UF : 1, UT : 1,		CONFIG : 'N U T, 0, 0, 1',
	X =  157.000  mm,	Y =  118.000  mm,	Z =   15.000 mm,
	W =180.000 deg,	P =   0.000 deg,	R =    90.000 deg
};
P[6139]{
   GP1:
	UF : 1, UT : 1,		CONFIG : 'N U T, 0, 0, 1',
	X =  160.000  mm,	Y =  118.000  mm,	Z =   15.000 mm,
	W =180.000 deg,	P =   0.000 deg,	R =    90.000 deg
};
P[6140]{
   GP1:
	UF : 1, UT : 1,		CONFIG : 'N U T, 0, 0, 1',
	X =  160.000  mm,	Y =  118.000  mm,	Z =   0.600 mm,
	W =180.000 deg,	P =   0.000 deg,	R =    90.000 deg
};
P[6141]{
   GP1:
	UF : 1, UT : 1,		CONFIG : 'N U T, 0, 0, 1',
	X =  160.000  mm,	Y =  118.000  mm,	Z =   15.000 mm,
	W =180.000 deg,	P =   0.000 deg,	R =    90.000 deg
};
P[6142]{
   GP1:
	UF : 1, UT : 1,		CONFIG : 'N U T, 0, 0, 1',
	X =  163.000  mm,	Y =  118.000  mm,	Z =   15.000 mm,
	W =180.000 deg,	P =   0.000 deg,	R =    90.000 deg
};
P[6143]{
   GP1:
	UF : 1, UT : 1,		CONFIG : 'N U T, 0, 0, 1',
	X =  163.000  mm,	Y =  118.000  mm,	Z =   0.600 mm,
	W =180.000 deg,	P =   0.000 deg,	R =    90.000 deg
};
P[6144]{
   GP1:
	UF : 1, UT : 1,		CONFIG : 'N U T, 0, 0, 1',
	X =  163.000  mm,	Y =  118.000  mm,	Z =   15.000 mm,
	W =180.000 deg,	P =   0.000 deg,	R =    90.000 deg
};
P[6145]{
   GP1:
	UF : 1, UT : 1,		CONFIG : 'N U T, 0, 0, 1',
	X =  166.000  mm,	Y =  118.000  mm,	Z =   15.000 mm,
	W =180.000 deg,	P =   0.000 deg,	R =    90.000 deg
};
P[6146]{
   GP1:
	UF : 1, UT : 1,		CONFIG : 'N U T, 0, 0, 1',
	X =  166.000  mm,	Y =  118.000  mm,	Z =   0.600 mm,
	W =180.000 deg,	P =   0.000 deg,	R =    90.000 deg
};
P[6147]{
   GP1:
	UF : 1, UT : 1,		CONFIG : 'N U T, 0, 0, 1',
	X =  166.000  mm,	Y =  118.000  mm,	Z =   15.000 mm,
	W =180.000 deg,	P =   0.000 deg,	R =    90.000 deg
};
P[6148]{
   GP1:
	UF : 1, UT : 1,		CONFIG : 'N U T, 0, 0, 1',
	X =  169.000  mm,	Y =  118.000  mm,	Z =   15.000 mm,
	W =180.000 deg,	P =   0.000 deg,	R =    90.000 deg
};
P[6149]{
   GP1:
	UF : 1, UT : 1,		CONFIG : 'N U T, 0, 0, 1',
	X =  169.000  mm,	Y =  118.000  mm,	Z =   0.600 mm,
	W =180.000 deg,	P =   0.000 deg,	R =    90.000 deg
};
P[6150]{
   GP1:
	UF : 1, UT : 1,		CONFIG : 'N U T, 0, 0, 1',
	X =  169.000  mm,	Y =  118.000  mm,	Z =   15.000 mm,
	W =180.000 deg,	P =   0.000 deg,	R =    90.000 deg
};
P[6151]{
   GP1:
	UF : 1, UT : 1,		CONFIG : 'N U T, 0, 0, 1',
	X =  172.000  mm,	Y =  118.000  mm,	Z =   15.000 mm,
	W =180.000 deg,	P =   0.000 deg,	R =    90.000 deg
};
P[6152]{
   GP1:
	UF : 1, UT : 1,		CONFIG : 'N U T, 0, 0, 1',
	X =  172.000  mm,	Y =  118.000  mm,	Z =   0.600 mm,
	W =180.000 deg,	P =   0.000 deg,	R =    90.000 deg
};
P[6153]{
   GP1:
	UF : 1, UT : 1,		CONFIG : 'N U T, 0, 0, 1',
	X =  172.000  mm,	Y =  118.000  mm,	Z =   15.000 mm,
	W =180.000 deg,	P =   0.000 deg,	R =    90.000 deg
};
P[6154]{
   GP1:
	UF : 1, UT : 1,		CONFIG : 'N U T, 0, 0, 1',
	X =  175.000  mm,	Y =  118.000  mm,	Z =   15.000 mm,
	W =180.000 deg,	P =   0.000 deg,	R =    90.000 deg
};
P[6155]{
   GP1:
	UF : 1, UT : 1,		CONFIG : 'N U T, 0, 0, 1',
	X =  175.000  mm,	Y =  118.000  mm,	Z =   0.600 mm,
	W =180.000 deg,	P =   0.000 deg,	R =    90.000 deg
};
P[6156]{
   GP1:
	UF : 1, UT : 1,		CONFIG : 'N U T, 0, 0, 1',
	X =  175.000  mm,	Y =  118.000  mm,	Z =   15.000 mm,
	W =180.000 deg,	P =   0.000 deg,	R =    90.000 deg
};
P[6157]{
   GP1:
	UF : 1, UT : 1,		CONFIG : 'N U T, 0, 0, 1',
	X =  178.000  mm,	Y =  118.000  mm,	Z =   15.000 mm,
	W =180.000 deg,	P =   0.000 deg,	R =    90.000 deg
};
P[6158]{
   GP1:
	UF : 1, UT : 1,		CONFIG : 'N U T, 0, 0, 1',
	X =  178.000  mm,	Y =  118.000  mm,	Z =   0.600 mm,
	W =180.000 deg,	P =   0.000 deg,	R =    90.000 deg
};
P[6159]{
   GP1:
	UF : 1, UT : 1,		CONFIG : 'N U T, 0, 0, 1',
	X =  178.000  mm,	Y =  118.000  mm,	Z =   15.000 mm,
	W =180.000 deg,	P =   0.000 deg,	R =    90.000 deg
};
P[6178]{
   GP1:
	UF : 1, UT : 1,		CONFIG : 'N U T, 0, 0, 1',
	X =  34.000  mm,	Y =  121.000  mm,	Z =   15.000 mm,
	W =180.000 deg,	P =   0.000 deg,	R =    90.000 deg
};
P[6179]{
   GP1:
	UF : 1, UT : 1,		CONFIG : 'N U T, 0, 0, 1',
	X =  34.000  mm,	Y =  121.000  mm,	Z =   0.600 mm,
	W =180.000 deg,	P =   0.000 deg,	R =    90.000 deg
};
P[6180]{
   GP1:
	UF : 1, UT : 1,		CONFIG : 'N U T, 0, 0, 1',
	X =  34.000  mm,	Y =  121.000  mm,	Z =   15.000 mm,
	W =180.000 deg,	P =   0.000 deg,	R =    90.000 deg
};
P[6181]{
   GP1:
	UF : 1, UT : 1,		CONFIG : 'N U T, 0, 0, 1',
	X =  37.000  mm,	Y =  121.000  mm,	Z =   15.000 mm,
	W =180.000 deg,	P =   0.000 deg,	R =    90.000 deg
};
P[6182]{
   GP1:
	UF : 1, UT : 1,		CONFIG : 'N U T, 0, 0, 1',
	X =  37.000  mm,	Y =  121.000  mm,	Z =   0.600 mm,
	W =180.000 deg,	P =   0.000 deg,	R =    90.000 deg
};
P[6183]{
   GP1:
	UF : 1, UT : 1,		CONFIG : 'N U T, 0, 0, 1',
	X =  37.000  mm,	Y =  121.000  mm,	Z =   15.000 mm,
	W =180.000 deg,	P =   0.000 deg,	R =    90.000 deg
};
P[6184]{
   GP1:
	UF : 1, UT : 1,		CONFIG : 'N U T, 0, 0, 1',
	X =  40.000  mm,	Y =  121.000  mm,	Z =   15.000 mm,
	W =180.000 deg,	P =   0.000 deg,	R =    90.000 deg
};
P[6185]{
   GP1:
	UF : 1, UT : 1,		CONFIG : 'N U T, 0, 0, 1',
	X =  40.000  mm,	Y =  121.000  mm,	Z =   0.600 mm,
	W =180.000 deg,	P =   0.000 deg,	R =    90.000 deg
};
P[6186]{
   GP1:
	UF : 1, UT : 1,		CONFIG : 'N U T, 0, 0, 1',
	X =  40.000  mm,	Y =  121.000  mm,	Z =   15.000 mm,
	W =180.000 deg,	P =   0.000 deg,	R =    90.000 deg
};
P[6211]{
   GP1:
	UF : 1, UT : 1,		CONFIG : 'N U T, 0, 0, 1',
	X =  115.000  mm,	Y =  121.000  mm,	Z =   15.000 mm,
	W =180.000 deg,	P =   0.000 deg,	R =    90.000 deg
};
P[6212]{
   GP1:
	UF : 1, UT : 1,		CONFIG : 'N U T, 0, 0, 1',
	X =  115.000  mm,	Y =  121.000  mm,	Z =   0.600 mm,
	W =180.000 deg,	P =   0.000 deg,	R =    90.000 deg
};
P[6213]{
   GP1:
	UF : 1, UT : 1,		CONFIG : 'N U T, 0, 0, 1',
	X =  115.000  mm,	Y =  121.000  mm,	Z =   15.000 mm,
	W =180.000 deg,	P =   0.000 deg,	R =    90.000 deg
};
P[6214]{
   GP1:
	UF : 1, UT : 1,		CONFIG : 'N U T, 0, 0, 1',
	X =  118.000  mm,	Y =  121.000  mm,	Z =   15.000 mm,
	W =180.000 deg,	P =   0.000 deg,	R =    90.000 deg
};
P[6215]{
   GP1:
	UF : 1, UT : 1,		CONFIG : 'N U T, 0, 0, 1',
	X =  118.000  mm,	Y =  121.000  mm,	Z =   0.600 mm,
	W =180.000 deg,	P =   0.000 deg,	R =    90.000 deg
};
P[6216]{
   GP1:
	UF : 1, UT : 1,		CONFIG : 'N U T, 0, 0, 1',
	X =  118.000  mm,	Y =  121.000  mm,	Z =   15.000 mm,
	W =180.000 deg,	P =   0.000 deg,	R =    90.000 deg
};
P[6217]{
   GP1:
	UF : 1, UT : 1,		CONFIG : 'N U T, 0, 0, 1',
	X =  121.000  mm,	Y =  121.000  mm,	Z =   15.000 mm,
	W =180.000 deg,	P =   0.000 deg,	R =    90.000 deg
};
P[6218]{
   GP1:
	UF : 1, UT : 1,		CONFIG : 'N U T, 0, 0, 1',
	X =  121.000  mm,	Y =  121.000  mm,	Z =   0.600 mm,
	W =180.000 deg,	P =   0.000 deg,	R =    90.000 deg
};
P[6219]{
   GP1:
	UF : 1, UT : 1,		CONFIG : 'N U T, 0, 0, 1',
	X =  121.000  mm,	Y =  121.000  mm,	Z =   15.000 mm,
	W =180.000 deg,	P =   0.000 deg,	R =    90.000 deg
};
P[6220]{
   GP1:
	UF : 1, UT : 1,		CONFIG : 'N U T, 0, 0, 1',
	X =  124.000  mm,	Y =  121.000  mm,	Z =   15.000 mm,
	W =180.000 deg,	P =   0.000 deg,	R =    90.000 deg
};
P[6221]{
   GP1:
	UF : 1, UT : 1,		CONFIG : 'N U T, 0, 0, 1',
	X =  124.000  mm,	Y =  121.000  mm,	Z =   0.600 mm,
	W =180.000 deg,	P =   0.000 deg,	R =    90.000 deg
};
P[6222]{
   GP1:
	UF : 1, UT : 1,		CONFIG : 'N U T, 0, 0, 1',
	X =  124.000  mm,	Y =  121.000  mm,	Z =   15.000 mm,
	W =180.000 deg,	P =   0.000 deg,	R =    90.000 deg
};
P[6223]{
   GP1:
	UF : 1, UT : 1,		CONFIG : 'N U T, 0, 0, 1',
	X =  127.000  mm,	Y =  121.000  mm,	Z =   15.000 mm,
	W =180.000 deg,	P =   0.000 deg,	R =    90.000 deg
};
P[6224]{
   GP1:
	UF : 1, UT : 1,		CONFIG : 'N U T, 0, 0, 1',
	X =  127.000  mm,	Y =  121.000  mm,	Z =   0.600 mm,
	W =180.000 deg,	P =   0.000 deg,	R =    90.000 deg
};
P[6225]{
   GP1:
	UF : 1, UT : 1,		CONFIG : 'N U T, 0, 0, 1',
	X =  127.000  mm,	Y =  121.000  mm,	Z =   15.000 mm,
	W =180.000 deg,	P =   0.000 deg,	R =    90.000 deg
};
P[6232]{
   GP1:
	UF : 1, UT : 1,		CONFIG : 'N U T, 0, 0, 1',
	X =  136.000  mm,	Y =  121.000  mm,	Z =   15.000 mm,
	W =180.000 deg,	P =   0.000 deg,	R =    90.000 deg
};
P[6233]{
   GP1:
	UF : 1, UT : 1,		CONFIG : 'N U T, 0, 0, 1',
	X =  136.000  mm,	Y =  121.000  mm,	Z =   0.600 mm,
	W =180.000 deg,	P =   0.000 deg,	R =    90.000 deg
};
P[6234]{
   GP1:
	UF : 1, UT : 1,		CONFIG : 'N U T, 0, 0, 1',
	X =  136.000  mm,	Y =  121.000  mm,	Z =   15.000 mm,
	W =180.000 deg,	P =   0.000 deg,	R =    90.000 deg
};
P[6235]{
   GP1:
